ACTION TEST_CASE_3_EXEC:
                        IF vTestCases[2].state = utTestCaseStates.ut_RUNNING THEN
	(*Run the test case*)
	IF NOT assertGreaterEqual_DINT(vTestCase3_act, vTestCase3_xp) THEN
		vTestCases[2].state := utTestCaseStates.ut_PASSED;
		vTestCases[2].msg := 'Parameter act was less than xp and function returned FALSE -> PASS';
	ELSE
		vTestCases[2].state := utTestCaseStates.ut_FAILED;
		vTestCases[2].msg := 'Parameter act was less than xp and function returned TRUE -> FAIL';
	END_IF
END_IF
                      
END_ACTION
END_PROGRAM

PROGRAM test_assertGreaterEqual_LWORD
  VAR
    vTestCases : ARRAY[0..20] OF utTestCase;  (* Definition of all test cases for this POU *)
    testRunner : utTestSuite;  (* Test Suite fb instance to run the tests *)
    vRunAll : BOOL;  (* Manual command to run all tests for this POU *)
    vResetAll : BOOL;  (* Manual command to reset all tests for this POU *)
    vTestCase1_act : LWORD;  (* Test data 1 of test case 1 *)
    vTestCase1_xp : LWORD;  (* Test data 2 of test case 1 *)
    vTestCase2_act : LWORD;  (* Test data 1 of test case 2 *)
    vTestCase2_xp : LWORD;  (* Test data 2 of test case 2 *)
    vTestCase3_act : LWORD;  (* Test data 1 of test case 3 *)
    vTestCase3_xp : LWORD;  (* Test data 2 of test case 3 *)
  END_VAR

                    (*Run the test cases*)
TEST_CASE_1_SETUP();
TEST_CASE_1_EXEC();

TEST_CASE_2_SETUP();
TEST_CASE_2_EXEC();

TEST_CASE_3_SETUP();
TEST_CASE_3_EXEC();

(*Instantiate the test runner*)
testRunner(
	Id := 75,
	Name := 'assertGreaterEqual_LWORD',
    RunTests := GVL.RunAll OR vRunAll,
	ResetTests := GVL.ResetAll OR vResetAll,
	TestCases:=vTestCases);

(*Report the results to the collection global*)
GVL.Results[testRunner.Id] := testRunner.Summary;
                  

ACTION TEST_CASE_1_EXEC:
                        IF vTestCases[0].state = utTestCaseStates.ut_RUNNING THEN
	(*Run the test case*)
	IF assertGreaterEqual_LWORD(vTestCase1_act, vTestCase1_xp) THEN
		vTestCases[0].state := utTestCaseStates.ut_PASSED;
		vTestCases[0].msg := 'Parameter act was greater than xp and function returned TRUE -> PASS';
	ELSE
		vTestCases[0].state := utTestCaseStates.ut_FAILED;
		vTestCases[0].msg := 'Parameter act was greater than xp and function returned FALSE -> FAIL';
	END_IF
END_IF
                      
END_ACTION

ACTION TEST_CASE_3_EXEC:
                        IF vTestCases[2].state = utTestCaseStates.ut_RUNNING THEN
	(*Run the test case*)
	IF NOT assertGreaterEqual_LWORD(vTestCase3_act, vTestCase3_xp) THEN
		vTestCases[2].state := utTestCaseStates.ut_PASSED;
		vTestCases[2].msg := 'Parameter act was less than xp and function returned FALSE -> PASS';
	ELSE
		vTestCases[2].state := utTestCaseStates.ut_FAILED;
		vTestCases[2].msg := 'Parameter act was less than xp and function returned TRUE -> FAIL';
	END_IF
END_IF
                      
END_ACTION

ACTION TEST_CASE_1_SETUP:
                        IF vTestCases[0].state = utTestCaseStates.ut_SETUP THEN
	(*Setup the test case information*)
	vTestCases[0].id := 1;
	vTestCases[0].desc[0] := 'RETURNS TRUE WHEN PARAMETER ACT GREATER THAN XP';
    vTestCases[0].desc[1] := 'Tests if the function returns True if the parameter act is greater than parameter xp';
	vTestCases[0].desc[2] := 'PASS IF: Return value is TRUE';
	
	(*Setup needed variables*)
	vTestCase1_act := REAL_TO_LWORD(115.4);
	vTestCase1_xp := REAL_TO_LWORD(85.4);
END_IF
                      
END_ACTION

ACTION TEST_CASE_2_SETUP:
                        IF vTestCases[1].state = utTestCaseStates.ut_SETUP THEN
	(*Setup the test case information*)
	vTestCases[1].id := 2;
    vTestCases[1].desc[0] := 'RETURNS TRUE WHEN PARAMETER ACT EQUAL TO XP';
    vTestCases[1].desc[1] := 'Tests if the function returns True if the parameter act is equal to parameter xp';
	vTestCases[1].desc[2] := 'PASS IF: Return value is TRUE';
	
	(*Setup needed variables*)
	vTestCase2_act := REAL_TO_LWORD(115.4);
	vTestCase2_xp := REAL_TO_LWORD(115.4);
END_IF
                      
END_ACTION

ACTION TEST_CASE_2_EXEC:
                        IF vTestCases[1].state = utTestCaseStates.ut_RUNNING THEN
	(*Run the test case*)
	IF assertGreaterEqual_LWORD(vTestCase2_act, vTestCase2_xp) THEN
		vTestCases[1].state := utTestCaseStates.ut_PASSED;
		vTestCases[1].msg := 'Parameter act was equal to xp and function returned TRUE -> PASS';
	ELSE
		vTestCases[1].state := utTestCaseStates.ut_FAILED;
		vTestCases[1].msg := 'Parameter act was equal to xp and function returned FALSE -> FAIL';
	END_IF
END_IF
                      
END_ACTION

ACTION TEST_CASE_3_SETUP:
                        IF vTestCases[2].state = utTestCaseStates.ut_SETUP THEN
	(*Setup the test case information*)
	vTestCases[2].id := 3;
    vTestCases[2].desc[0] := 'RETURNS FALSE WHEN PARAMETER ACT LESS THAN XP';
    vTestCases[2].desc[1] := 'Tests if the function returns False if the parameter act is less than parameter xp';
	vTestCases[2].desc[2] := 'PASS IF: Return value is FALSE';
	
	(*Setup needed variables*)
	vTestCase3_act := REAL_TO_LWORD(85.4);
	vTestCase3_xp := REAL_TO_LWORD(115.4);
END_IF
                      
END_ACTION
END_PROGRAM

PROGRAM test_assertGreaterEqual_ULINT
  VAR
    vTestCases : ARRAY[0..20] OF utTestCase;  (* Definition of all test cases for this POU *)
    testRunner : utTestSuite;  (* Test Suite fb instance to run the tests *)
    vRunAll : BOOL;  (* Manual command to run all tests for this POU *)
    vResetAll : BOOL;  (* Manual command to reset all tests for this POU *)
    vTestCase1_act : ULINT;  (* Test data 1 of test case 1 *)
    vTestCase1_xp : ULINT;  (* Test data 2 of test case 1 *)
    vTestCase2_act : ULINT;  (* Test data 1 of test case 2 *)
    vTestCase2_xp : ULINT;  (* Test data 2 of test case 2 *)
    vTestCase3_act : ULINT;  (* Test data 1 of test case 3 *)
    vTestCase3_xp : ULINT;  (* Test data 2 of test case 3 *)
  END_VAR

                    (*Run the test cases*)
TEST_CASE_1_SETUP();
TEST_CASE_1_EXEC();

TEST_CASE_2_SETUP();
TEST_CASE_2_EXEC();

TEST_CASE_3_SETUP();
TEST_CASE_3_EXEC();

(*Instantiate the test runner*)
testRunner(
	Id := 83,
	Name := 'assertGreaterEqual_ULINT',
    RunTests := GVL.RunAll OR vRunAll,
	ResetTests := GVL.ResetAll OR vResetAll,
	TestCases:=vTestCases);

(*Report the results to the collection global*)
GVL.Results[testRunner.Id] := testRunner.Summary;
                  

ACTION TEST_CASE_2_EXEC:
                        IF vTestCases[1].state = utTestCaseStates.ut_RUNNING THEN
	(*Run the test case*)
	IF assertGreaterEqual_ULINT(vTestCase2_act, vTestCase2_xp) THEN
		vTestCases[1].state := utTestCaseStates.ut_PASSED;
		vTestCases[1].msg := 'Parameter act was equal to xp and function returned TRUE -> PASS';
	ELSE
		vTestCases[1].state := utTestCaseStates.ut_FAILED;
		vTestCases[1].msg := 'Parameter act was equal to xp and function returned FALSE -> FAIL';
	END_IF
END_IF
                      
END_ACTION

ACTION TEST_CASE_1_SETUP:
                        IF vTestCases[0].state = utTestCaseStates.ut_SETUP THEN
	(*Setup the test case information*)
	vTestCases[0].id := 1;
	vTestCases[0].desc[0] := 'RETURNS TRUE WHEN PARAMETER ACT GREATER THAN XP';
    vTestCases[0].desc[1] := 'Tests if the function returns True if the parameter act is greater than parameter xp';
	vTestCases[0].desc[2] := 'PASS IF: Return value is TRUE';
	
	(*Setup needed variables*)
	vTestCase1_act := REAL_TO_ULINT(115.4);
	vTestCase1_xp := REAL_TO_ULINT(85.4);
END_IF
                      
END_ACTION

ACTION TEST_CASE_1_EXEC:
                        IF vTestCases[0].state = utTestCaseStates.ut_RUNNING THEN
	(*Run the test case*)
	IF assertGreaterEqual_ULINT(vTestCase1_act, vTestCase1_xp) THEN
		vTestCases[0].state := utTestCaseStates.ut_PASSED;
		vTestCases[0].msg := 'Parameter act was greater than xp and function returned TRUE -> PASS';
	ELSE
		vTestCases[0].state := utTestCaseStates.ut_FAILED;
		vTestCases[0].msg := 'Parameter act was greater than xp and function returned FALSE -> FAIL';
	END_IF
END_IF
                      
END_ACTION

ACTION TEST_CASE_2_SETUP:
                        IF vTestCases[1].state = utTestCaseStates.ut_SETUP THEN
	(*Setup the test case information*)
	vTestCases[1].id := 2;
    vTestCases[1].desc[0] := 'RETURNS TRUE WHEN PARAMETER ACT EQUAL TO XP';
    vTestCases[1].desc[1] := 'Tests if the function returns True if the parameter act is equal to parameter xp';
	vTestCases[1].desc[2] := 'PASS IF: Return value is TRUE';
	
	(*Setup needed variables*)
	vTestCase2_act := REAL_TO_ULINT(115.4);
	vTestCase2_xp := REAL_TO_ULINT(115.4);
END_IF
                      
END_ACTION

ACTION TEST_CASE_3_SETUP:
                        IF vTestCases[2].state = utTestCaseStates.ut_SETUP THEN
	(*Setup the test case information*)
	vTestCases[2].id := 3;
    vTestCases[2].desc[0] := 'RETURNS FALSE WHEN PARAMETER ACT LESS THAN XP';
    vTestCases[2].desc[1] := 'Tests if the function returns False if the parameter act is less than parameter xp';
	vTestCases[2].desc[2] := 'PASS IF: Return value is FALSE';
	
	(*Setup needed variables*)
	vTestCase3_act := REAL_TO_ULINT(85.4);
	vTestCase3_xp := REAL_TO_ULINT(115.4);
END_IF
                      
END_ACTION

ACTION TEST_CASE_3_EXEC:
                        IF vTestCases[2].state = utTestCaseStates.ut_RUNNING THEN
	(*Run the test case*)
	IF NOT assertGreaterEqual_ULINT(vTestCase3_act, vTestCase3_xp) THEN
		vTestCases[2].state := utTestCaseStates.ut_PASSED;
		vTestCases[2].msg := 'Parameter act was less than xp and function returned FALSE -> PASS';
	ELSE
		vTestCases[2].state := utTestCaseStates.ut_FAILED;
		vTestCases[2].msg := 'Parameter act was less than xp and function returned TRUE -> FAIL';
	END_IF
END_IF
                      
END_ACTION
END_PROGRAM

PROGRAM test_assertGreaterEqual_SINT
  VAR
    vTestCases : ARRAY[0..20] OF utTestCase;  (* Definition of all test cases for this POU *)
    testRunner : utTestSuite;  (* Test Suite fb instance to run the tests *)
    vRunAll : BOOL;  (* Manual command to run all tests for this POU *)
    vResetAll : BOOL;  (* Manual command to reset all tests for this POU *)
    vTestCase1_act : SINT;  (* Test data 1 of test case 1 *)
    vTestCase1_xp : SINT;  (* Test data 2 of test case 1 *)
    vTestCase2_act : SINT;  (* Test data 1 of test case 2 *)
    vTestCase2_xp : SINT;  (* Test data 2 of test case 2 *)
    vTestCase3_act : SINT;  (* Test data 1 of test case 3 *)
    vTestCase3_xp : SINT;  (* Test data 2 of test case 3 *)
  END_VAR

                    (*Run the test cases*)
TEST_CASE_1_SETUP();
TEST_CASE_1_EXEC();

TEST_CASE_2_SETUP();
TEST_CASE_2_EXEC();

TEST_CASE_3_SETUP();
TEST_CASE_3_EXEC();

(*Instantiate the test runner*)
testRunner(
	Id := 76,
	Name := 'assertGreaterEqual_SINT',
    RunTests := GVL.RunAll OR vRunAll,
	ResetTests := GVL.ResetAll OR vResetAll,
	TestCases:=vTestCases);

(*Report the results to the collection global*)
GVL.Results[testRunner.Id] := testRunner.Summary;
                  

ACTION TEST_CASE_2_EXEC:
                        IF vTestCases[1].state = utTestCaseStates.ut_RUNNING THEN
	(*Run the test case*)
	IF assertGreaterEqual_SINT(vTestCase2_act, vTestCase2_xp) THEN
		vTestCases[1].state := utTestCaseStates.ut_PASSED;
		vTestCases[1].msg := 'Parameter act was equal to xp and function returned TRUE -> PASS';
	ELSE
		vTestCases[1].state := utTestCaseStates.ut_FAILED;
		vTestCases[1].msg := 'Parameter act was equal to xp and function returned FALSE -> FAIL';
	END_IF
END_IF
                      
END_ACTION

ACTION TEST_CASE_1_SETUP:
                        IF vTestCases[0].state = utTestCaseStates.ut_SETUP THEN
	(*Setup the test case information*)
	vTestCases[0].id := 1;
	vTestCases[0].desc[0] := 'RETURNS TRUE WHEN PARAMETER ACT GREATER THAN XP';
    vTestCases[0].desc[1] := 'Tests if the function returns True if the parameter act is greater than parameter xp';
	vTestCases[0].desc[2] := 'PASS IF: Return value is TRUE';
	
	(*Setup needed variables*)
	vTestCase1_act := REAL_TO_SINT(115.4);
	vTestCase1_xp := REAL_TO_SINT(85.4);
END_IF
                      
END_ACTION

ACTION TEST_CASE_1_EXEC:
                        IF vTestCases[0].state = utTestCaseStates.ut_RUNNING THEN
	(*Run the test case*)
	IF assertGreaterEqual_SINT(vTestCase1_act, vTestCase1_xp) THEN
		vTestCases[0].state := utTestCaseStates.ut_PASSED;
		vTestCases[0].msg := 'Parameter act was greater than xp and function returned TRUE -> PASS';
	ELSE
		vTestCases[0].state := utTestCaseStates.ut_FAILED;
		vTestCases[0].msg := 'Parameter act was greater than xp and function returned FALSE -> FAIL';
	END_IF
END_IF
                      
END_ACTION

ACTION TEST_CASE_2_SETUP:
                        IF vTestCases[1].state = utTestCaseStates.ut_SETUP THEN
	(*Setup the test case information*)
	vTestCases[1].id := 2;
    vTestCases[1].desc[0] := 'RETURNS TRUE WHEN PARAMETER ACT EQUAL TO XP';
    vTestCases[1].desc[1] := 'Tests if the function returns True if the parameter act is equal to parameter xp';
	vTestCases[1].desc[2] := 'PASS IF: Return value is TRUE';
	
	(*Setup needed variables*)
	vTestCase2_act := REAL_TO_SINT(115.4);
	vTestCase2_xp := REAL_TO_SINT(115.4);
END_IF
                      
END_ACTION

ACTION TEST_CASE_3_SETUP:
                        IF vTestCases[2].state = utTestCaseStates.ut_SETUP THEN
	(*Setup the test case information*)
	vTestCases[2].id := 3;
    vTestCases[2].desc[0] := 'RETURNS FALSE WHEN PARAMETER ACT LESS THAN XP';
    vTestCases[2].desc[1] := 'Tests if the function returns False if the parameter act is less than parameter xp';
	vTestCases[2].desc[2] := 'PASS IF: Return value is FALSE';
	
	(*Setup needed variables*)
	vTestCase3_act := REAL_TO_SINT(85.4);
	vTestCase3_xp := REAL_TO_SINT(115.4);
END_IF
                      
END_ACTION

ACTION TEST_CASE_3_EXEC:
                        IF vTestCases[2].state = utTestCaseStates.ut_RUNNING THEN
	(*Run the test case*)
	IF NOT assertGreaterEqual_SINT(vTestCase3_act, vTestCase3_xp) THEN
		vTestCases[2].state := utTestCaseStates.ut_PASSED;
		vTestCases[2].msg := 'Parameter act was less than xp and function returned FALSE -> PASS';
	ELSE
		vTestCases[2].state := utTestCaseStates.ut_FAILED;
		vTestCases[2].msg := 'Parameter act was less than xp and function returned TRUE -> FAIL';
	END_IF
END_IF
                      
END_ACTION
END_PROGRAM

PROGRAM test_assertGreater_LREAL
  VAR
    vTestCases : ARRAY[0..20] OF utTestCase;  (* Definition of all test cases for this POU *)
    testRunner : utTestSuite;  (* Test Suite fb instance to run the tests *)
    vRunAll : BOOL;  (* Manual command to run all tests for this POU *)
    vResetAll : BOOL;  (* Manual command to reset all tests for this POU *)
    vTestCase1_act : LREAL;  (* Test data 1 of test case 1 *)
    vTestCase1_xp : LREAL;  (* Test data 2 of test case 1 *)
    vTestCase2_act : LREAL;  (* Test data 1 of test case 2 *)
    vTestCase2_xp : LREAL;  (* Test data 2 of test case 2 *)
  END_VAR

                    (*Run the test cases*)
TEST_CASE_1_SETUP();
TEST_CASE_1_EXEC();

TEST_CASE_2_SETUP();
TEST_CASE_2_EXEC();

(*Instantiate the test runner*)
testRunner(
	Id := 63,
	Name := 'assertGreater_LREAL',
    RunTests := GVL.RunAll OR vRunAll,
	ResetTests := GVL.ResetAll OR vResetAll,
	TestCases:=vTestCases);

(*Report the results to the collection global*)
GVL.Results[testRunner.Id] := testRunner.Summary;
                  

ACTION TEST_CASE_1_SETUP:
                        IF vTestCases[0].state = utTestCaseStates.ut_SETUP THEN
	(*Setup the test case information*)
	vTestCases[0].id := 1;
	vTestCases[0].desc[0] := 'RETURNS TRUE WHEN PARAMETER ACT GREATER THAN XP';
    vTestCases[0].desc[1] := 'Tests if the function returns True if the parameter act is greater than parameter xp';
	vTestCases[0].desc[2] := 'PASS IF: Return value is TRUE';
	
	(*Setup needed variables*)
	vTestCase1_act := REAL_TO_LREAL(115.4);
	vTestCase1_xp := REAL_TO_LREAL(85.4);
END_IF
                      
END_ACTION

ACTION TEST_CASE_1_EXEC:
                        IF vTestCases[0].state = utTestCaseStates.ut_RUNNING THEN
	(*Run the test case*)
	IF assertGreater_LREAL(vTestCase1_act, vTestCase1_xp) THEN
		vTestCases[0].state := utTestCaseStates.ut_PASSED;
		vTestCases[0].msg := 'Parameter act was greater than xp and function returned TRUE -> PASS';
	ELSE
		vTestCases[0].state := utTestCaseStates.ut_FAILED;
		vTestCases[0].msg := 'Parameter act was greater than xp and function returned FALSE -> FAIL';
	END_IF
END_IF
                      
END_ACTION

ACTION TEST_CASE_2_SETUP:
                        IF vTestCases[1].state = utTestCaseStates.ut_SETUP THEN
	(*Setup the test case information*)
	vTestCases[1].id := 2;
    vTestCases[1].desc[0] := 'RETURNS FALSE WHEN PARAMETER ACT LESS THAN XP';
    vTestCases[1].desc[1] := 'Tests if the function returns False if the parameter act is less than parameter xp';
	vTestCases[1].desc[2] := 'PASS IF: Return value is FALSE';
	
	(*Setup needed variables*)
	vTestCase2_act := REAL_TO_LREAL(8.4);
	vTestCase2_xp := REAL_TO_LREAL(85.4);
END_IF
                      
END_ACTION

ACTION TEST_CASE_2_EXEC:
                        IF vTestCases[1].state = utTestCaseStates.ut_RUNNING THEN
	(*Run the test case*)
	IF NOT assertGreater_LREAL(vTestCase2_act, vTestCase2_xp) THEN
		vTestCases[1].state := utTestCaseStates.ut_PASSED;
		vTestCases[1].msg := 'Parameter act was less than xp and function returned FALSE -> PASS';
	ELSE
		vTestCases[1].state := utTestCaseStates.ut_FAILED;
		vTestCases[1].msg := 'Parameter act was less than xp and function returned TRUE -> FAIL';
	END_IF
END_IF
                      
END_ACTION
END_PROGRAM

PROGRAM test_assertGreater_TIME
  VAR
    vTestCases : ARRAY[0..20] OF utTestCase;  (* Definition of all test cases for this POU *)
    testRunner : utTestSuite;  (* Test Suite fb instance to run the tests *)
    vRunAll : BOOL;  (* Manual command to run all tests for this POU *)
    vResetAll : BOOL;  (* Manual command to reset all tests for this POU *)
    vTestCase1_act : TIME;  (* Test data 1 of test case 1 *)
    vTestCase1_xp : TIME;  (* Test data 2 of test case 1 *)
    vTestCase2_act : TIME;  (* Test data 1 of test case 2 *)
    vTestCase2_xp : TIME;  (* Test data 2 of test case 2 *)
  END_VAR

                    (*Run the test cases*)
TEST_CASE_1_SETUP();
TEST_CASE_1_EXEC();

TEST_CASE_2_SETUP();
TEST_CASE_2_EXEC();

(*Instantiate the test runner*)
testRunner(
	Id := 64,
	Name := 'assertGreater_TIME',
    RunTests := GVL.RunAll OR vRunAll,
	ResetTests := GVL.ResetAll OR vResetAll,
	TestCases:=vTestCases);

(*Report the results to the collection global*)
GVL.Results[testRunner.Id] := testRunner.Summary;
                  

ACTION TEST_CASE_1_SETUP:
                        IF vTestCases[0].state = utTestCaseStates.ut_SETUP THEN
	(*Setup the test case information*)
	vTestCases[0].id := 1;
	vTestCases[0].desc[0] := 'RETURNS TRUE WHEN PARAMETER ACT GREATER THAN XP';
    vTestCases[0].desc[1] := 'Tests if the function returns True if the parameter act is greater than parameter xp';
	vTestCases[0].desc[2] := 'PASS IF: Return value is TRUE';
	
	(*Setup needed variables*)
	vTestCase1_act := REAL_TO_TIME(115.4);
	vTestCase1_xp := REAL_TO_TIME(85.4);
END_IF
                      
END_ACTION

ACTION TEST_CASE_1_EXEC:
                        IF vTestCases[0].state = utTestCaseStates.ut_RUNNING THEN
	(*Run the test case*)
	IF assertGreater_TIME(vTestCase1_act, vTestCase1_xp) THEN
		vTestCases[0].state := utTestCaseStates.ut_PASSED;
		vTestCases[0].msg := 'Parameter act was greater than xp and function returned TRUE -> PASS';
	ELSE
		vTestCases[0].state := utTestCaseStates.ut_FAILED;
		vTestCases[0].msg := 'Parameter act was greater than xp and function returned FALSE -> FAIL';
	END_IF
END_IF
                      
END_ACTION

ACTION TEST_CASE_2_SETUP:
                        IF vTestCases[1].state = utTestCaseStates.ut_SETUP THEN
	(*Setup the test case information*)
	vTestCases[1].id := 2;
    vTestCases[1].desc[0] := 'RETURNS FALSE WHEN PARAMETER ACT LESS THAN XP';
    vTestCases[1].desc[1] := 'Tests if the function returns False if the parameter act is less than parameter xp';
	vTestCases[1].desc[2] := 'PASS IF: Return value is FALSE';
	
	(*Setup needed variables*)
	vTestCase2_act := REAL_TO_TIME(8.4);
	vTestCase2_xp := REAL_TO_TIME(85.4);
END_IF
                      
END_ACTION

ACTION TEST_CASE_2_EXEC:
                        IF vTestCases[1].state = utTestCaseStates.ut_RUNNING THEN
	(*Run the test case*)
	IF NOT assertGreater_TIME(vTestCase2_act, vTestCase2_xp) THEN
		vTestCases[1].state := utTestCaseStates.ut_PASSED;
		vTestCases[1].msg := 'Parameter act was less than xp and function returned FALSE -> PASS';
	ELSE
		vTestCases[1].state := utTestCaseStates.ut_FAILED;
		vTestCases[1].msg := 'Parameter act was less than xp and function returned TRUE -> FAIL';
	END_IF
END_IF
                      
END_ACTION
END_PROGRAM

PROGRAM test_assertGreater_TIME_OF_DAY
  VAR
    vTestCases : ARRAY[0..20] OF utTestCase;  (* Definition of all test cases for this POU *)
    testRunner : utTestSuite;  (* Test Suite fb instance to run the tests *)
    vRunAll : BOOL;  (* Manual command to run all tests for this POU *)
    vResetAll : BOOL;  (* Manual command to reset all tests for this POU *)
    vTestCase1_act : TOD;  (* Test data 1 of test case 1 *)
    vTestCase1_xp : TOD;  (* Test data 2 of test case 1 *)
    vTestCase2_act : TOD;  (* Test data 1 of test case 2 *)
    vTestCase2_xp : TOD;  (* Test data 2 of test case 2 *)
  END_VAR

                    (*Run the test cases*)
TEST_CASE_1_SETUP();
TEST_CASE_1_EXEC();

TEST_CASE_2_SETUP();
TEST_CASE_2_EXEC();

(*Instantiate the test runner*)
testRunner(
	Id := 70,
	Name := 'assertGreater_TIME_OF_DAY',
    RunTests := GVL.RunAll OR vRunAll,
	ResetTests := GVL.ResetAll OR vResetAll,
	TestCases:=vTestCases);

(*Report the results to the collection global*)
GVL.Results[testRunner.Id] := testRunner.Summary;
                  

ACTION TEST_CASE_1_SETUP:
                        IF vTestCases[0].state = utTestCaseStates.ut_SETUP THEN
	(*Setup the test case information*)
	vTestCases[0].id := 1;
	vTestCases[0].desc[0] := 'RETURNS TRUE WHEN PARAMETER ACT GREATER THAN XP';
    vTestCases[0].desc[1] := 'Tests if the function returns True if the parameter act is greater than parameter xp';
	vTestCases[0].desc[2] := 'PASS IF: Return value is TRUE';
	
	(*Setup needed variables*)
	vTestCase1_act := REAL_TO_TOD(115.4);
	vTestCase1_xp := REAL_TO_TOD(85.4);
END_IF
                      
END_ACTION

ACTION TEST_CASE_1_EXEC:
                        IF vTestCases[0].state = utTestCaseStates.ut_RUNNING THEN
	(*Run the test case*)
	IF assertGreater_TIME_OF_DAY(vTestCase1_act, vTestCase1_xp) THEN
		vTestCases[0].state := utTestCaseStates.ut_PASSED;
		vTestCases[0].msg := 'Parameter act was greater than xp and function returned TRUE -> PASS';
	ELSE
		vTestCases[0].state := utTestCaseStates.ut_FAILED;
		vTestCases[0].msg := 'Parameter act was greater than xp and function returned FALSE -> FAIL';
	END_IF
END_IF
                      
END_ACTION

ACTION TEST_CASE_2_SETUP:
                        IF vTestCases[1].state = utTestCaseStates.ut_SETUP THEN
	(*Setup the test case information*)
	vTestCases[1].id := 2;
    vTestCases[1].desc[0] := 'RETURNS FALSE WHEN PARAMETER ACT LESS THAN XP';
    vTestCases[1].desc[1] := 'Tests if the function returns False if the parameter act is less than parameter xp';
	vTestCases[1].desc[2] := 'PASS IF: Return value is FALSE';
	
	(*Setup needed variables*)
	vTestCase2_act := REAL_TO_TOD(8.4);
	vTestCase2_xp := REAL_TO_TOD(85.4);
END_IF
                      
END_ACTION

ACTION TEST_CASE_2_EXEC:
                        IF vTestCases[1].state = utTestCaseStates.ut_RUNNING THEN
	(*Run the test case*)
	IF NOT assertGreater_TIME_OF_DAY(vTestCase2_act, vTestCase2_xp) THEN
		vTestCases[1].state := utTestCaseStates.ut_PASSED;
		vTestCases[1].msg := 'Parameter act was less than xp and function returned FALSE -> PASS';
	ELSE
		vTestCases[1].state := utTestCaseStates.ut_FAILED;
		vTestCases[1].msg := 'Parameter act was less than xp and function returned TRUE -> FAIL';
	END_IF
END_IF
                      
END_ACTION
END_PROGRAM

PROGRAM test_assertGreater_LTIME_OF_DAY
  VAR
    vTestCases : ARRAY[0..20] OF utTestCase;  (* Definition of all test cases for this POU *)
    testRunner : utTestSuite;  (* Test Suite fb instance to run the tests *)
    vRunAll : BOOL;  (* Manual command to run all tests for this POU *)
    vResetAll : BOOL;  (* Manual command to reset all tests for this POU *)
    vTestCase1_act : LTIME_OF_DAY;  (* Test data 1 of test case 1 *)
    vTestCase1_xp : LTIME_OF_DAY;  (* Test data 2 of test case 1 *)
    vTestCase2_act : LTIME_OF_DAY;  (* Test data 1 of test case 2 *)
    vTestCase2_xp : LTIME_OF_DAY;  (* Test data 2 of test case 2 *)
  END_VAR

                    (*Run the test cases*)
TEST_CASE_1_SETUP();
TEST_CASE_1_EXEC();

TEST_CASE_2_SETUP();
TEST_CASE_2_EXEC();

(*Instantiate the test runner*)
testRunner(
	Id := 71,
	Name := 'assertGreater_LTIME_OF_DAY',
    RunTests := GVL.RunAll OR vRunAll,
	ResetTests := GVL.ResetAll OR vResetAll,
	TestCases:=vTestCases);

(*Report the results to the collection global*)
GVL.Results[testRunner.Id] := testRunner.Summary;
                  

ACTION TEST_CASE_1_SETUP:
                        IF vTestCases[0].state = utTestCaseStates.ut_SETUP THEN
	(*Setup the test case information*)
	vTestCases[0].id := 1;
	vTestCases[0].desc[0] := 'RETURNS TRUE WHEN PARAMETER ACT GREATER THAN XP';
    vTestCases[0].desc[1] := 'Tests if the function returns True if the parameter act is greater than parameter xp';
	vTestCases[0].desc[2] := 'PASS IF: Return value is TRUE';
	
	(*Setup needed variables*)
	vTestCase1_act := REAL_TO_LTOD(115.4);
	vTestCase1_xp := REAL_TO_LTOD(85.4);
END_IF
                      
END_ACTION

ACTION TEST_CASE_1_EXEC:
                        IF vTestCases[0].state = utTestCaseStates.ut_RUNNING THEN
	(*Run the test case*)
	IF assertGreater_LTIME_OF_DAY(vTestCase1_act, vTestCase1_xp) THEN
		vTestCases[0].state := utTestCaseStates.ut_PASSED;
		vTestCases[0].msg := 'Parameter act was greater than xp and function returned TRUE -> PASS';
	ELSE
		vTestCases[0].state := utTestCaseStates.ut_FAILED;
		vTestCases[0].msg := 'Parameter act was greater than xp and function returned FALSE -> FAIL';
	END_IF
END_IF
                      
END_ACTION

ACTION TEST_CASE_2_SETUP:
                        IF vTestCases[1].state = utTestCaseStates.ut_SETUP THEN
	(*Setup the test case information*)
	vTestCases[1].id := 2;
    vTestCases[1].desc[0] := 'RETURNS FALSE WHEN PARAMETER ACT LESS THAN XP';
    vTestCases[1].desc[1] := 'Tests if the function returns False if the parameter act is less than parameter xp';
	vTestCases[1].desc[2] := 'PASS IF: Return value is FALSE';
	
	(*Setup needed variables*)
	vTestCase2_act := REAL_TO_LTOD(8.4);
	vTestCase2_xp := REAL_TO_LTOD(85.4);
END_IF
                      
END_ACTION

ACTION TEST_CASE_2_EXEC:
                        IF vTestCases[1].state = utTestCaseStates.ut_RUNNING THEN
	(*Run the test case*)
	IF NOT assertGreater_LTIME_OF_DAY(vTestCase2_act, vTestCase2_xp) THEN
		vTestCases[1].state := utTestCaseStates.ut_PASSED;
		vTestCases[1].msg := 'Parameter act was less than xp and function returned FALSE -> PASS';
	ELSE
		vTestCases[1].state := utTestCaseStates.ut_FAILED;
		vTestCases[1].msg := 'Parameter act was less than xp and function returned TRUE -> FAIL';
	END_IF
END_IF
                      
END_ACTION
END_PROGRAM

PROGRAM test_assertGreater_LTIME
  VAR
    vTestCases : ARRAY[0..20] OF utTestCase;  (* Definition of all test cases for this POU *)
    testRunner : utTestSuite;  (* Test Suite fb instance to run the tests *)
    vRunAll : BOOL;  (* Manual command to run all tests for this POU *)
    vResetAll : BOOL;  (* Manual command to reset all tests for this POU *)
    vTestCase1_act : LTIME;  (* Test data 1 of test case 1 *)
    vTestCase1_xp : LTIME;  (* Test data 2 of test case 1 *)
    vTestCase2_act : LTIME;  (* Test data 1 of test case 2 *)
    vTestCase2_xp : LTIME;  (* Test data 2 of test case 2 *)
  END_VAR

                    (*Run the test cases*)
TEST_CASE_1_SETUP();
TEST_CASE_1_EXEC();

TEST_CASE_2_SETUP();
TEST_CASE_2_EXEC();

(*Instantiate the test runner*)
testRunner(
	Id := 65,
	Name := 'assertGreater_LTIME',
    RunTests := GVL.RunAll OR vRunAll,
	ResetTests := GVL.ResetAll OR vResetAll,
	TestCases:=vTestCases);

(*Report the results to the collection global*)
GVL.Results[testRunner.Id] := testRunner.Summary;
                  

ACTION TEST_CASE_2_SETUP:
                        IF vTestCases[1].state = utTestCaseStates.ut_SETUP THEN
	(*Setup the test case information*)
	vTestCases[1].id := 2;
    vTestCases[1].desc[0] := 'RETURNS FALSE WHEN PARAMETER ACT LESS THAN XP';
    vTestCases[1].desc[1] := 'Tests if the function returns False if the parameter act is less than parameter xp';
	vTestCases[1].desc[2] := 'PASS IF: Return value is FALSE';
	
	(*Setup needed variables*)
	vTestCase2_act := REAL_TO_LTIME(8.4);
	vTestCase2_xp := REAL_TO_LTIME(85.4);
END_IF
                      
END_ACTION

ACTION TEST_CASE_2_EXEC:
                        IF vTestCases[1].state = utTestCaseStates.ut_RUNNING THEN
	(*Run the test case*)
	IF NOT assertGreater_LTIME(vTestCase2_act, vTestCase2_xp) THEN
		vTestCases[1].state := utTestCaseStates.ut_PASSED;
		vTestCases[1].msg := 'Parameter act was less than xp and function returned FALSE -> PASS';
	ELSE
		vTestCases[1].state := utTestCaseStates.ut_FAILED;
		vTestCases[1].msg := 'Parameter act was less than xp and function returned TRUE -> FAIL';
	END_IF
END_IF
                      
END_ACTION

ACTION TEST_CASE_1_SETUP:
                        IF vTestCases[0].state = utTestCaseStates.ut_SETUP THEN
	(*Setup the test case information*)
	vTestCases[0].id := 1;
	vTestCases[0].desc[0] := 'RETURNS TRUE WHEN PARAMETER ACT GREATER THAN XP';
    vTestCases[0].desc[1] := 'Tests if the function returns True if the parameter act is greater than parameter xp';
	vTestCases[0].desc[2] := 'PASS IF: Return value is TRUE';
	
	(*Setup needed variables*)
	vTestCase1_act := REAL_TO_LTIME(115.4);
	vTestCase1_xp := REAL_TO_LTIME(85.4);
END_IF
                      
END_ACTION

ACTION TEST_CASE_1_EXEC:
                        IF vTestCases[0].state = utTestCaseStates.ut_RUNNING THEN
	(*Run the test case*)
	IF assertGreater_LTIME(vTestCase1_act, vTestCase1_xp) THEN
		vTestCases[0].state := utTestCaseStates.ut_PASSED;
		vTestCases[0].msg := 'Parameter act was greater than xp and function returned TRUE -> PASS';
	ELSE
		vTestCases[0].state := utTestCaseStates.ut_FAILED;
		vTestCases[0].msg := 'Parameter act was greater than xp and function returned FALSE -> FAIL';
	END_IF
END_IF
                      
END_ACTION
END_PROGRAM

PROGRAM test_assertGreaterEqual_BYTE
  VAR
    vTestCases : ARRAY[0..20] OF utTestCase;  (* Definition of all test cases for this POU *)
    testRunner : utTestSuite;  (* Test Suite fb instance to run the tests *)
    vRunAll : BOOL;  (* Manual command to run all tests for this POU *)
    vResetAll : BOOL;  (* Manual command to reset all tests for this POU *)
    vTestCase1_act : BYTE;  (* Test data 1 of test case 1 *)
    vTestCase1_xp : BYTE;  (* Test data 2 of test case 1 *)
    vTestCase2_act : BYTE;  (* Test data 1 of test case 2 *)
    vTestCase2_xp : BYTE;  (* Test data 2 of test case 2 *)
    vTestCase3_act : BYTE;  (* Test data 1 of test case 3 *)
    vTestCase3_xp : BYTE;  (* Test data 2 of test case 3 *)
  END_VAR

                    (*Run the test cases*)
TEST_CASE_1_SETUP();
TEST_CASE_1_EXEC();

TEST_CASE_2_SETUP();
TEST_CASE_2_EXEC();

TEST_CASE_3_SETUP();
TEST_CASE_3_EXEC();

(*Instantiate the test runner*)
testRunner(
	Id := 72,
	Name := 'assertGreaterEqual_BYTE',
    RunTests := GVL.RunAll OR vRunAll,
	ResetTests := GVL.ResetAll OR vResetAll,
	TestCases:=vTestCases);

(*Report the results to the collection global*)
GVL.Results[testRunner.Id] := testRunner.Summary;
                  

ACTION TEST_CASE_2_SETUP:
                        IF vTestCases[1].state = utTestCaseStates.ut_SETUP THEN
	(*Setup the test case information*)
	vTestCases[1].id := 2;
    vTestCases[1].desc[0] := 'RETURNS TRUE WHEN PARAMETER ACT EQUAL TO XP';
    vTestCases[1].desc[1] := 'Tests if the function returns True if the parameter act is equal to parameter xp';
	vTestCases[1].desc[2] := 'PASS IF: Return value is TRUE';
	
	(*Setup needed variables*)
	vTestCase2_act := REAL_TO_BYTE(115.4);
	vTestCase2_xp := REAL_TO_BYTE(115.4);
END_IF
                      
END_ACTION

ACTION TEST_CASE_3_SETUP:
                        IF vTestCases[2].state = utTestCaseStates.ut_SETUP THEN
	(*Setup the test case information*)
	vTestCases[2].id := 3;
    vTestCases[2].desc[0] := 'RETURNS FALSE WHEN PARAMETER ACT LESS THAN XP';
    vTestCases[2].desc[1] := 'Tests if the function returns False if the parameter act is less than parameter xp';
	vTestCases[2].desc[2] := 'PASS IF: Return value is FALSE';
	
	(*Setup needed variables*)
	vTestCase3_act := REAL_TO_BYTE(85.4);
	vTestCase3_xp := REAL_TO_BYTE(115.4);
END_IF
                      
END_ACTION

ACTION TEST_CASE_2_EXEC:
                        IF vTestCases[1].state = utTestCaseStates.ut_RUNNING THEN
	(*Run the test case*)
	IF assertGreaterEqual_BYTE(vTestCase2_act, vTestCase2_xp) THEN
		vTestCases[1].state := utTestCaseStates.ut_PASSED;
		vTestCases[1].msg := 'Parameter act was equal to xp and function returned TRUE -> PASS';
	ELSE
		vTestCases[1].state := utTestCaseStates.ut_FAILED;
		vTestCases[1].msg := 'Parameter act was equal to xp and function returned FALSE -> FAIL';
	END_IF
END_IF
                      
END_ACTION

ACTION TEST_CASE_1_SETUP:
                        IF vTestCases[0].state = utTestCaseStates.ut_SETUP THEN
	(*Setup the test case information*)
	vTestCases[0].id := 1;
	vTestCases[0].desc[0] := 'RETURNS TRUE WHEN PARAMETER ACT GREATER THAN XP';
    vTestCases[0].desc[1] := 'Tests if the function returns True if the parameter act is greater than parameter xp';
	vTestCases[0].desc[2] := 'PASS IF: Return value is TRUE';
	
	(*Setup needed variables*)
	vTestCase1_act := REAL_TO_BYTE(115.4);
	vTestCase1_xp := REAL_TO_BYTE(85.4);
END_IF
                      
END_ACTION

ACTION TEST_CASE_1_EXEC:
                        IF vTestCases[0].state = utTestCaseStates.ut_RUNNING THEN
	(*Run the test case*)
	IF assertGreaterEqual_BYTE(vTestCase1_act, vTestCase1_xp) THEN
		vTestCases[0].state := utTestCaseStates.ut_PASSED;
		vTestCases[0].msg := 'Parameter act was greater than xp and function returned TRUE -> PASS';
	ELSE
		vTestCases[0].state := utTestCaseStates.ut_FAILED;
		vTestCases[0].msg := 'Parameter act was greater than xp and function returned FALSE -> FAIL';
	END_IF
END_IF
                      
END_ACTION

ACTION TEST_CASE_3_EXEC:
                        IF vTestCases[2].state = utTestCaseStates.ut_RUNNING THEN
	(*Run the test case*)
	IF NOT assertGreaterEqual_BYTE(vTestCase3_act, vTestCase3_xp) THEN
		vTestCases[2].state := utTestCaseStates.ut_PASSED;
		vTestCases[2].msg := 'Parameter act was less than xp and function returned FALSE -> PASS';
	ELSE
		vTestCases[2].state := utTestCaseStates.ut_FAILED;
		vTestCases[2].msg := 'Parameter act was less than xp and function returned TRUE -> FAIL';
	END_IF
END_IF
                      
END_ACTION
END_PROGRAM

PROGRAM test_assertGreaterEqual_REAL
  VAR
    vTestCases : ARRAY[0..20] OF utTestCase;  (* Definition of all test cases for this POU *)
    testRunner : utTestSuite;  (* Test Suite fb instance to run the tests *)
    vRunAll : BOOL;  (* Manual command to run all tests for this POU *)
    vResetAll : BOOL;  (* Manual command to reset all tests for this POU *)
    vTestCase1_act : REAL;  (* Test data 1 of test case 1 *)
    vTestCase1_xp : REAL;  (* Test data 2 of test case 1 *)
    vTestCase2_act : REAL;  (* Test data 1 of test case 2 *)
    vTestCase2_xp : REAL;  (* Test data 2 of test case 2 *)
    vTestCase3_act : REAL;  (* Test data 1 of test case 3 *)
    vTestCase3_xp : REAL;  (* Test data 2 of test case 3 *)
  END_VAR

                    (*Run the test cases*)
TEST_CASE_1_SETUP();
TEST_CASE_1_EXEC();

TEST_CASE_2_SETUP();
TEST_CASE_2_EXEC();

TEST_CASE_3_SETUP();
TEST_CASE_3_EXEC();

(*Instantiate the test runner*)
testRunner(
	Id := 84,
	Name := 'assertGreaterEqual_REAL',
    RunTests := GVL.RunAll OR vRunAll,
	ResetTests := GVL.ResetAll OR vResetAll,
	TestCases:=vTestCases);

(*Report the results to the collection global*)
GVL.Results[testRunner.Id] := testRunner.Summary;
                  

ACTION TEST_CASE_1_SETUP:
                        IF vTestCases[0].state = utTestCaseStates.ut_SETUP THEN
	(*Setup the test case information*)
	vTestCases[0].id := 1;
	vTestCases[0].desc[0] := 'RETURNS TRUE WHEN PARAMETER ACT GREATER THAN XP';
    vTestCases[0].desc[1] := 'Tests if the function returns True if the parameter act is greater than parameter xp';
	vTestCases[0].desc[2] := 'PASS IF: Return value is TRUE';
	
	(*Setup needed variables*)
	vTestCase1_act := 115.4;
	vTestCase1_xp := 85.4;
END_IF
                      
END_ACTION

ACTION TEST_CASE_1_EXEC:
                        IF vTestCases[0].state = utTestCaseStates.ut_RUNNING THEN
	(*Run the test case*)
	IF assertGreaterEqual_REAL(vTestCase1_act, vTestCase1_xp) THEN
		vTestCases[0].state := utTestCaseStates.ut_PASSED;
		vTestCases[0].msg := 'Parameter act was greater than xp and function returned TRUE -> PASS';
	ELSE
		vTestCases[0].state := utTestCaseStates.ut_FAILED;
		vTestCases[0].msg := 'Parameter act was greater than xp and function returned FALSE -> FAIL';
	END_IF
END_IF
                      
END_ACTION

ACTION TEST_CASE_2_SETUP:
                        IF vTestCases[1].state = utTestCaseStates.ut_SETUP THEN
	(*Setup the test case information*)
	vTestCases[1].id := 2;
    vTestCases[1].desc[0] := 'RETURNS TRUE WHEN PARAMETER ACT EQUAL TO XP';
    vTestCases[1].desc[1] := 'Tests if the function returns True if the parameter act is equal to parameter xp';
	vTestCases[1].desc[2] := 'PASS IF: Return value is TRUE';
	
	(*Setup needed variables*)
	vTestCase2_act := 115.4;
	vTestCase2_xp := 115.4;
END_IF
                      
END_ACTION

ACTION TEST_CASE_2_EXEC:
                        IF vTestCases[1].state = utTestCaseStates.ut_RUNNING THEN
	(*Run the test case*)
	IF assertGreaterEqual_REAL(vTestCase2_act, vTestCase2_xp) THEN
		vTestCases[1].state := utTestCaseStates.ut_PASSED;
		vTestCases[1].msg := 'Parameter act was equal to xp and function returned TRUE -> PASS';
	ELSE
		vTestCases[1].state := utTestCaseStates.ut_FAILED;
		vTestCases[1].msg := 'Parameter act was equal to xp and function returned FALSE -> FAIL';
	END_IF
END_IF
                      
END_ACTION

ACTION TEST_CASE_3_SETUP:
                        IF vTestCases[2].state = utTestCaseStates.ut_SETUP THEN
	(*Setup the test case information*)
	vTestCases[2].id := 3;
    vTestCases[2].desc[0] := 'RETURNS FALSE WHEN PARAMETER ACT LESS THAN XP';
    vTestCases[2].desc[1] := 'Tests if the function returns False if the parameter act is less than parameter xp';
	vTestCases[2].desc[2] := 'PASS IF: Return value is FALSE';
	
	(*Setup needed variables*)
	vTestCase3_act := 85.4;
	vTestCase3_xp := 115.4;
END_IF
                      
END_ACTION

ACTION TEST_CASE_3_EXEC:
                        IF vTestCases[2].state = utTestCaseStates.ut_RUNNING THEN
	(*Run the test case*)
	IF NOT assertGreaterEqual_REAL(vTestCase3_act, vTestCase3_xp) THEN
		vTestCases[2].state := utTestCaseStates.ut_PASSED;
		vTestCases[2].msg := 'Parameter act was less than xp and function returned FALSE -> PASS';
	ELSE
		vTestCases[2].state := utTestCaseStates.ut_FAILED;
		vTestCases[2].msg := 'Parameter act was less than xp and function returned TRUE -> FAIL';
	END_IF
END_IF
                      
END_ACTION
END_PROGRAM

PROGRAM test_assertGreaterEqual_LREAL
  VAR
    vTestCases : ARRAY[0..20] OF utTestCase;  (* Definition of all test cases for this POU *)
    testRunner : utTestSuite;  (* Test Suite fb instance to run the tests *)
    vRunAll : BOOL;  (* Manual command to run all tests for this POU *)
    vResetAll : BOOL;  (* Manual command to reset all tests for this POU *)
    vTestCase1_act : LREAL;  (* Test data 1 of test case 1 *)
    vTestCase1_xp : LREAL;  (* Test data 2 of test case 1 *)
    vTestCase2_act : LREAL;  (* Test data 1 of test case 2 *)
    vTestCase2_xp : LREAL;  (* Test data 2 of test case 2 *)
    vTestCase3_act : LREAL;  (* Test data 1 of test case 3 *)
    vTestCase3_xp : LREAL;  (* Test data 2 of test case 3 *)
  END_VAR

                    (*Run the test cases*)
TEST_CASE_1_SETUP();
TEST_CASE_1_EXEC();

TEST_CASE_2_SETUP();
TEST_CASE_2_EXEC();

TEST_CASE_3_SETUP();
TEST_CASE_3_EXEC();

(*Instantiate the test runner*)
testRunner(
	Id := 85,
	Name := 'assertGreaterEqual_LREAL',
    RunTests := GVL.RunAll OR vRunAll,
	ResetTests := GVL.ResetAll OR vResetAll,
	TestCases:=vTestCases);

(*Report the results to the collection global*)
GVL.Results[testRunner.Id] := testRunner.Summary;
                  

ACTION TEST_CASE_1_SETUP:
                        IF vTestCases[0].state = utTestCaseStates.ut_SETUP THEN
	(*Setup the test case information*)
	vTestCases[0].id := 1;
	vTestCases[0].desc[0] := 'RETURNS TRUE WHEN PARAMETER ACT GREATER THAN XP';
    vTestCases[0].desc[1] := 'Tests if the function returns True if the parameter act is greater than parameter xp';
	vTestCases[0].desc[2] := 'PASS IF: Return value is TRUE';
	
	(*Setup needed variables*)
	vTestCase1_act := REAL_TO_LREAL(115.4);
	vTestCase1_xp := REAL_TO_LREAL(85.4);
END_IF
                      
END_ACTION

ACTION TEST_CASE_1_EXEC:
                        IF vTestCases[0].state = utTestCaseStates.ut_RUNNING THEN
	(*Run the test case*)
	IF assertGreaterEqual_LREAL(vTestCase1_act, vTestCase1_xp) THEN
		vTestCases[0].state := utTestCaseStates.ut_PASSED;
		vTestCases[0].msg := 'Parameter act was greater than xp and function returned TRUE -> PASS';
	ELSE
		vTestCases[0].state := utTestCaseStates.ut_FAILED;
		vTestCases[0].msg := 'Parameter act was greater than xp and function returned FALSE -> FAIL';
	END_IF
END_IF
                      
END_ACTION

ACTION TEST_CASE_2_SETUP:
                        IF vTestCases[1].state = utTestCaseStates.ut_SETUP THEN
	(*Setup the test case information*)
	vTestCases[1].id := 2;
    vTestCases[1].desc[0] := 'RETURNS TRUE WHEN PARAMETER ACT EQUAL TO XP';
    vTestCases[1].desc[1] := 'Tests if the function returns True if the parameter act is equal to parameter xp';
	vTestCases[1].desc[2] := 'PASS IF: Return value is TRUE';
	
	(*Setup needed variables*)
	vTestCase2_act := REAL_TO_LREAL(115.4);
	vTestCase2_xp := REAL_TO_LREAL(115.4);
END_IF
                      
END_ACTION

ACTION TEST_CASE_2_EXEC:
                        IF vTestCases[1].state = utTestCaseStates.ut_RUNNING THEN
	(*Run the test case*)
	IF assertGreaterEqual_LREAL(vTestCase2_act, vTestCase2_xp) THEN
		vTestCases[1].state := utTestCaseStates.ut_PASSED;
		vTestCases[1].msg := 'Parameter act was equal to xp and function returned TRUE -> PASS';
	ELSE
		vTestCases[1].state := utTestCaseStates.ut_FAILED;
		vTestCases[1].msg := 'Parameter act was equal to xp and function returned FALSE -> FAIL';
	END_IF
END_IF
                      
END_ACTION

ACTION TEST_CASE_3_SETUP:
                        IF vTestCases[2].state = utTestCaseStates.ut_SETUP THEN
	(*Setup the test case information*)
	vTestCases[2].id := 3;
    vTestCases[2].desc[0] := 'RETURNS FALSE WHEN PARAMETER ACT LESS THAN XP';
    vTestCases[2].desc[1] := 'Tests if the function returns False if the parameter act is less than parameter xp';
	vTestCases[2].desc[2] := 'PASS IF: Return value is FALSE';
	
	(*Setup needed variables*)
	vTestCase3_act := REAL_TO_LREAL(85.4);
	vTestCase3_xp := REAL_TO_LREAL(115.4);
END_IF
                      
END_ACTION

ACTION TEST_CASE_3_EXEC:
                        IF vTestCases[2].state = utTestCaseStates.ut_RUNNING THEN
	(*Run the test case*)
	IF NOT assertGreaterEqual_LREAL(vTestCase3_act, vTestCase3_xp) THEN
		vTestCases[2].state := utTestCaseStates.ut_PASSED;
		vTestCases[2].msg := 'Parameter act was less than xp and function returned FALSE -> PASS';
	ELSE
		vTestCases[2].state := utTestCaseStates.ut_FAILED;
		vTestCases[2].msg := 'Parameter act was less than xp and function returned TRUE -> FAIL';
	END_IF
END_IF
                      
END_ACTION
END_PROGRAM

PROGRAM test_assertGreaterEqual_USINT
  VAR
    vTestCases : ARRAY[0..20] OF utTestCase;  (* Definition of all test cases for this POU *)
    testRunner : utTestSuite;  (* Test Suite fb instance to run the tests *)
    vRunAll : BOOL;  (* Manual command to run all tests for this POU *)
    vResetAll : BOOL;  (* Manual command to reset all tests for this POU *)
    vTestCase1_act : USINT;  (* Test data 1 of test case 1 *)
    vTestCase1_xp : USINT;  (* Test data 2 of test case 1 *)
    vTestCase2_act : USINT;  (* Test data 1 of test case 2 *)
    vTestCase2_xp : USINT;  (* Test data 2 of test case 2 *)
    vTestCase3_act : USINT;  (* Test data 1 of test case 3 *)
    vTestCase3_xp : USINT;  (* Test data 2 of test case 3 *)
  END_VAR

                    (*Run the test cases*)
TEST_CASE_1_SETUP();
TEST_CASE_1_EXEC();

TEST_CASE_2_SETUP();
TEST_CASE_2_EXEC();

TEST_CASE_3_SETUP();
TEST_CASE_3_EXEC();

(*Instantiate the test runner*)
testRunner(
	Id := 77,
	Name := 'assertGreaterEqual_USINT',
    RunTests := GVL.RunAll OR vRunAll,
	ResetTests := GVL.ResetAll OR vResetAll,
	TestCases:=vTestCases);

(*Report the results to the collection global*)
GVL.Results[testRunner.Id] := testRunner.Summary;
                  

ACTION TEST_CASE_1_SETUP:
                        IF vTestCases[0].state = utTestCaseStates.ut_SETUP THEN
	(*Setup the test case information*)
	vTestCases[0].id := 1;
	vTestCases[0].desc[0] := 'RETURNS TRUE WHEN PARAMETER ACT GREATER THAN XP';
    vTestCases[0].desc[1] := 'Tests if the function returns True if the parameter act is greater than parameter xp';
	vTestCases[0].desc[2] := 'PASS IF: Return value is TRUE';
	
	(*Setup needed variables*)
	vTestCase1_act := REAL_TO_USINT(115.4);
	vTestCase1_xp := REAL_TO_USINT(85.4);
END_IF
                      
END_ACTION

ACTION TEST_CASE_1_EXEC:
                        IF vTestCases[0].state = utTestCaseStates.ut_RUNNING THEN
	(*Run the test case*)
	IF assertGreaterEqual_USINT(vTestCase1_act, vTestCase1_xp) THEN
		vTestCases[0].state := utTestCaseStates.ut_PASSED;
		vTestCases[0].msg := 'Parameter act was greater than xp and function returned TRUE -> PASS';
	ELSE
		vTestCases[0].state := utTestCaseStates.ut_FAILED;
		vTestCases[0].msg := 'Parameter act was greater than xp and function returned FALSE -> FAIL';
	END_IF
END_IF
                      
END_ACTION

ACTION TEST_CASE_2_SETUP:
                        IF vTestCases[1].state = utTestCaseStates.ut_SETUP THEN
	(*Setup the test case information*)
	vTestCases[1].id := 2;
    vTestCases[1].desc[0] := 'RETURNS TRUE WHEN PARAMETER ACT EQUAL TO XP';
    vTestCases[1].desc[1] := 'Tests if the function returns True if the parameter act is equal to parameter xp';
	vTestCases[1].desc[2] := 'PASS IF: Return value is TRUE';
	
	(*Setup needed variables*)
	vTestCase2_act := REAL_TO_USINT(115.4);
	vTestCase2_xp := REAL_TO_USINT(115.4);
END_IF
                      
END_ACTION

ACTION TEST_CASE_2_EXEC:
                        IF vTestCases[1].state = utTestCaseStates.ut_RUNNING THEN
	(*Run the test case*)
	IF assertGreaterEqual_USINT(vTestCase2_act, vTestCase2_xp) THEN
		vTestCases[1].state := utTestCaseStates.ut_PASSED;
		vTestCases[1].msg := 'Parameter act was equal to xp and function returned TRUE -> PASS';
	ELSE
		vTestCases[1].state := utTestCaseStates.ut_FAILED;
		vTestCases[1].msg := 'Parameter act was equal to xp and function returned FALSE -> FAIL';
	END_IF
END_IF
                      
END_ACTION

ACTION TEST_CASE_3_SETUP:
                        IF vTestCases[2].state = utTestCaseStates.ut_SETUP THEN
	(*Setup the test case information*)
	vTestCases[2].id := 3;
    vTestCases[2].desc[0] := 'RETURNS FALSE WHEN PARAMETER ACT LESS THAN XP';
    vTestCases[2].desc[1] := 'Tests if the function returns False if the parameter act is less than parameter xp';
	vTestCases[2].desc[2] := 'PASS IF: Return value is FALSE';
	
	(*Setup needed variables*)
	vTestCase3_act := REAL_TO_USINT(85.4);
	vTestCase3_xp := REAL_TO_USINT(115.4);
END_IF
                      
END_ACTION

ACTION TEST_CASE_3_EXEC:
                        IF vTestCases[2].state = utTestCaseStates.ut_RUNNING THEN
	(*Run the test case*)
	IF NOT assertGreaterEqual_USINT(vTestCase3_act, vTestCase3_xp) THEN
		vTestCases[2].state := utTestCaseStates.ut_PASSED;
		vTestCases[2].msg := 'Parameter act was less than xp and function returned FALSE -> PASS';
	ELSE
		vTestCases[2].state := utTestCaseStates.ut_FAILED;
		vTestCases[2].msg := 'Parameter act was less than xp and function returned TRUE -> FAIL';
	END_IF
END_IF
                      
END_ACTION
END_PROGRAM

PROGRAM test_assertGreaterEqual_INT
  VAR
    vTestCases : ARRAY[0..20] OF utTestCase;  (* Definition of all test cases for this POU *)
    testRunner : utTestSuite;  (* Test Suite fb instance to run the tests *)
    vRunAll : BOOL;  (* Manual command to run all tests for this POU *)
    vResetAll : BOOL;  (* Manual command to reset all tests for this POU *)
    vTestCase1_act : INT;  (* Test data 1 of test case 1 *)
    vTestCase1_xp : INT;  (* Test data 2 of test case 1 *)
    vTestCase2_act : INT;  (* Test data 1 of test case 2 *)
    vTestCase2_xp : INT;  (* Test data 2 of test case 2 *)
    vTestCase3_act : INT;  (* Test data 1 of test case 3 *)
    vTestCase3_xp : INT;  (* Test data 2 of test case 3 *)
  END_VAR

                    (*Run the test cases*)
TEST_CASE_1_SETUP();
TEST_CASE_1_EXEC();

TEST_CASE_2_SETUP();
TEST_CASE_2_EXEC();

TEST_CASE_3_SETUP();
TEST_CASE_3_EXEC();

(*Instantiate the test runner*)
testRunner(
	Id := 78,
	Name := 'assertGreaterEqual_INT',
    RunTests := GVL.RunAll OR vRunAll,
	ResetTests := GVL.ResetAll OR vResetAll,
	TestCases:=vTestCases);

(*Report the results to the collection global*)
GVL.Results[testRunner.Id] := testRunner.Summary;
                  

ACTION TEST_CASE_1_SETUP:
                        IF vTestCases[0].state = utTestCaseStates.ut_SETUP THEN
	(*Setup the test case information*)
	vTestCases[0].id := 1;
	vTestCases[0].desc[0] := 'RETURNS TRUE WHEN PARAMETER ACT GREATER THAN XP';
    vTestCases[0].desc[1] := 'Tests if the function returns True if the parameter act is greater than parameter xp';
	vTestCases[0].desc[2] := 'PASS IF: Return value is TRUE';
	
	(*Setup needed variables*)
	vTestCase1_act := REAL_TO_INT(115.4);
	vTestCase1_xp := REAL_TO_INT(85.4);
END_IF
                      
END_ACTION

ACTION TEST_CASE_1_EXEC:
                        IF vTestCases[0].state = utTestCaseStates.ut_RUNNING THEN
	(*Run the test case*)
	IF assertGreaterEqual_INT(vTestCase1_act, vTestCase1_xp) THEN
		vTestCases[0].state := utTestCaseStates.ut_PASSED;
		vTestCases[0].msg := 'Parameter act was greater than xp and function returned TRUE -> PASS';
	ELSE
		vTestCases[0].state := utTestCaseStates.ut_FAILED;
		vTestCases[0].msg := 'Parameter act was greater than xp and function returned FALSE -> FAIL';
	END_IF
END_IF
                      
END_ACTION

ACTION TEST_CASE_2_SETUP:
                        IF vTestCases[1].state = utTestCaseStates.ut_SETUP THEN
	(*Setup the test case information*)
	vTestCases[1].id := 2;
    vTestCases[1].desc[0] := 'RETURNS TRUE WHEN PARAMETER ACT EQUAL TO XP';
    vTestCases[1].desc[1] := 'Tests if the function returns True if the parameter act is equal to parameter xp';
	vTestCases[1].desc[2] := 'PASS IF: Return value is TRUE';
	
	(*Setup needed variables*)
	vTestCase2_act := REAL_TO_INT(115.4);
	vTestCase2_xp := REAL_TO_INT(115.4);
END_IF
                      
END_ACTION

ACTION TEST_CASE_2_EXEC:
                        IF vTestCases[1].state = utTestCaseStates.ut_RUNNING THEN
	(*Run the test case*)
	IF assertGreaterEqual_INT(vTestCase2_act, vTestCase2_xp) THEN
		vTestCases[1].state := utTestCaseStates.ut_PASSED;
		vTestCases[1].msg := 'Parameter act was equal to xp and function returned TRUE -> PASS';
	ELSE
		vTestCases[1].state := utTestCaseStates.ut_FAILED;
		vTestCases[1].msg := 'Parameter act was equal to xp and function returned FALSE -> FAIL';
	END_IF
END_IF
                      
END_ACTION

ACTION TEST_CASE_3_SETUP:
                        IF vTestCases[2].state = utTestCaseStates.ut_SETUP THEN
	(*Setup the test case information*)
	vTestCases[2].id := 3;
    vTestCases[2].desc[0] := 'RETURNS FALSE WHEN PARAMETER ACT LESS THAN XP';
    vTestCases[2].desc[1] := 'Tests if the function returns False if the parameter act is less than parameter xp';
	vTestCases[2].desc[2] := 'PASS IF: Return value is FALSE';
	
	(*Setup needed variables*)
	vTestCase3_act := REAL_TO_INT(85.4);
	vTestCase3_xp := REAL_TO_INT(115.4);
END_IF
                      
END_ACTION

ACTION TEST_CASE_3_EXEC:
                        IF vTestCases[2].state = utTestCaseStates.ut_RUNNING THEN
	(*Run the test case*)
	IF NOT assertGreaterEqual_INT(vTestCase3_act, vTestCase3_xp) THEN
		vTestCases[2].state := utTestCaseStates.ut_PASSED;
		vTestCases[2].msg := 'Parameter act was less than xp and function returned FALSE -> PASS';
	ELSE
		vTestCases[2].state := utTestCaseStates.ut_FAILED;
		vTestCases[2].msg := 'Parameter act was less than xp and function returned TRUE -> FAIL';
	END_IF
END_IF
                      
END_ACTION
END_PROGRAM

PROGRAM test_assertArrayEqual_WSTRING
  VAR
    vTestCases : ARRAY[0..20] OF utTestCase;  (* Definition of all test cases for this POU *)
    testRunner : utTestSuite;  (* Test Suite fb instance to run the tests *)
    vRunAll : BOOL;  (* Manual command to run all tests for this POU *)
    vResetAll : BOOL;  (* Manual command to reset all tests for this POU *)
    vTestCase1_act : ARRAY[0..70] OF WSTRING;  (* Array data 1 of test case 1 *)
    vTestCase1_xp : ARRAY[0..70] OF WSTRING;  (* Array data 2 of test case 1 *)
    vTestCase2_act : ARRAY[0..70] OF WSTRING;  (* Array data 3 of test case 2 *)
    vTestCase2_xp : ARRAY[0..70] OF WSTRING;  (* Array data 4 of test case 2 *)
    i : UINT;  (* Iterator variable i *)
    j : UINT;  (* Iterator variable j *)
  END_VAR

                    (*Run the test cases*)
TEST_CASE_1_SETUP();
TEST_CASE_1_EXEC();

TEST_CASE_2_SETUP();
TEST_CASE_2_EXEC();

(*Instantiate the test runner*)
testRunner(
	Id := 154,
	Name := 'assertArrayEqual_WSTRING',
    RunTests := GVL.RunAll OR vRunAll,
	ResetTests := GVL.ResetAll OR vResetAll,
	TestCases:=vTestCases);

(*Report the results to the collection global*)
GVL.Results[testRunner.Id] := testRunner.Summary;
                  

ACTION TEST_CASE_1_SETUP:
                        IF vTestCases[0].state = utTestCaseStates.ut_SETUP THEN
	(*Setup the test case information*)
	vTestCases[0].id := 1;
	vTestCases[0].desc[0] := 'RETURNS TRUE WHEN ARRAYS EQUAL';
    vTestCases[0].desc[1] := 'Tests if the function returns True if the passed in arrays are identical';
	vTestCases[0].desc[2] := 'PASS IF: Return value is TRUE';
	
	(*Setup needed variables*)
	FOR i:=0 TO 70 DO
		vTestCase1_act[i] := UINT_TO_WSTRING(35 * BOOL_TO_UINT(i MOD 2 = 0));
		vTestCase1_xp[i] := UINT_TO_WSTRING(35 * BOOL_TO_UINT(i MOD 2 = 0));
	END_FOR
END_IF
                      
END_ACTION

ACTION TEST_CASE_1_EXEC:
                        IF vTestCases[0].state = utTestCaseStates.ut_RUNNING THEN
	(*Run the test case*)
	IF assertArrayEqual_WSTRING(ADR(vTestCase1_act), ADR(vTestCase1_xp), SIZEOF(vTestCase1_act)) THEN
		vTestCases[0].state := utTestCaseStates.ut_PASSED;
		vTestCases[0].msg := 'Arrays were equal and function returned TRUE -> PASS';
	ELSE
		vTestCases[0].state := utTestCaseStates.ut_FAILED;
		vTestCases[0].msg := 'Arrays were equal and function returned FALSE -> FAIL';
	END_IF
END_IF
                      
END_ACTION

ACTION TEST_CASE_2_SETUP:
                        IF vTestCases[1].state = utTestCaseStates.ut_SETUP THEN
	(*Setup the test case information*)
	vTestCases[1].id := 2;
	vTestCases[1].desc[0] := 'RETURNS FALSE WHEN ARRAYS NOT EQUAL';
    vTestCases[1].desc[1] := 'Tests if the function returns False if the passed in arrays are not identical';
	vTestCases[1].desc[2] := 'PASS IF: Return value is FALSE';
	
	(*Setup needed variables*)
	FOR j:=0 TO 70 DO
		vTestCase2_act[j] := UINT_TO_WSTRING(35 * BOOL_TO_UINT(j MOD 2 = 0));
		vTestCase2_xp[j] := UINT_TO_WSTRING(35 * BOOL_TO_UINT(j MOD 2 <> 0));
	END_FOR
END_IF
                      
END_ACTION

ACTION TEST_CASE_2_EXEC:
                        IF vTestCases[1].state = utTestCaseStates.ut_RUNNING THEN
	(*Run the test case*)
	IF NOT assertArrayEqual_WSTRING(ADR(vTestCase2_act), ADR(vTestCase2_xp), SIZEOF(vTestCase2_act)) THEN
		vTestCases[1].state := utTestCaseStates.ut_PASSED;
		vTestCases[1].msg := 'Arrays were not equal and function returned FALSE -> PASS';
	ELSE
		vTestCases[1].state := utTestCaseStates.ut_FAILED;
		vTestCases[1].msg := 'Arrays were not equal and function returned TRUE -> FAIL';
	END_IF
END_IF
                      
END_ACTION
END_PROGRAM

PROGRAM test_assertArrayEqual_TIME
  VAR
    vTestCases : ARRAY[0..20] OF utTestCase;  (* Definition of all test cases for this POU *)
    testRunner : utTestSuite;  (* Test Suite fb instance to run the tests *)
    vRunAll : BOOL;  (* Manual command to run all tests for this POU *)
    vResetAll : BOOL;  (* Manual command to reset all tests for this POU *)
    vTestCase1_act : ARRAY[0..70] OF TIME;  (* Array data 1 of test case 1 *)
    vTestCase1_xp : ARRAY[0..70] OF TIME;  (* Array data 2 of test case 1 *)
    vTestCase2_act : ARRAY[0..70] OF TIME;  (* Array data 3 of test case 2 *)
    vTestCase2_xp : ARRAY[0..70] OF TIME;  (* Array data 4 of test case 2 *)
    i : UINT;  (* Iterator variable i *)
    j : UINT;  (* Iterator variable j *)
  END_VAR

                    (*Run the test cases*)
TEST_CASE_1_SETUP();
TEST_CASE_1_EXEC();

TEST_CASE_2_SETUP();
TEST_CASE_2_EXEC();

(*Instantiate the test runner*)
testRunner(
	Id := 155,
	Name := 'assertArrayEqual_TIME',
    RunTests := GVL.RunAll OR vRunAll,
	ResetTests := GVL.ResetAll OR vResetAll,
	TestCases:=vTestCases);

(*Report the results to the collection global*)
GVL.Results[testRunner.Id] := testRunner.Summary;
                  

ACTION TEST_CASE_1_SETUP:
                        IF vTestCases[0].state = utTestCaseStates.ut_SETUP THEN
	(*Setup the test case information*)
	vTestCases[0].id := 1;
	vTestCases[0].desc[0] := 'RETURNS TRUE WHEN ARRAYS EQUAL';
    vTestCases[0].desc[1] := 'Tests if the function returns True if the passed in arrays are identical';
	vTestCases[0].desc[2] := 'PASS IF: Return value is TRUE';
	
	(*Setup needed variables*)
	FOR i:=0 TO 70 DO
		vTestCase1_act[i] := UINT_TO_TIME(35 * BOOL_TO_UINT(i MOD 2 = 0));
		vTestCase1_xp[i] := UINT_TO_TIME(35 * BOOL_TO_UINT(i MOD 2 = 0));
	END_FOR
END_IF
                      
END_ACTION

ACTION TEST_CASE_1_EXEC:
                        IF vTestCases[0].state = utTestCaseStates.ut_RUNNING THEN
	(*Run the test case*)
	IF assertArrayEqual_TIME(ADR(vTestCase1_act), ADR(vTestCase1_xp), SIZEOF(vTestCase1_act)) THEN
		vTestCases[0].state := utTestCaseStates.ut_PASSED;
		vTestCases[0].msg := 'Arrays were equal and function returned TRUE -> PASS';
	ELSE
		vTestCases[0].state := utTestCaseStates.ut_FAILED;
		vTestCases[0].msg := 'Arrays were equal and function returned FALSE -> FAIL';
	END_IF
END_IF
                      
END_ACTION

ACTION TEST_CASE_2_SETUP:
                        IF vTestCases[1].state = utTestCaseStates.ut_SETUP THEN
	(*Setup the test case information*)
	vTestCases[1].id := 2;
	vTestCases[1].desc[0] := 'RETURNS FALSE WHEN ARRAYS NOT EQUAL';
    vTestCases[1].desc[1] := 'Tests if the function returns False if the passed in arrays are not identical';
	vTestCases[1].desc[2] := 'PASS IF: Return value is FALSE';
	
	(*Setup needed variables*)
	FOR j:=0 TO 70 DO
		vTestCase2_act[j] := UINT_TO_TIME(35 * BOOL_TO_UINT(j MOD 2 = 0));
		vTestCase2_xp[j] := UINT_TO_TIME(35 * BOOL_TO_UINT(j MOD 2 <> 0));
	END_FOR
END_IF
                      
END_ACTION

ACTION TEST_CASE_2_EXEC:
                        IF vTestCases[1].state = utTestCaseStates.ut_RUNNING THEN
	(*Run the test case*)
	IF NOT assertArrayEqual_TIME(ADR(vTestCase2_act), ADR(vTestCase2_xp), SIZEOF(vTestCase2_act)) THEN
		vTestCases[1].state := utTestCaseStates.ut_PASSED;
		vTestCases[1].msg := 'Arrays were not equal and function returned FALSE -> PASS';
	ELSE
		vTestCases[1].state := utTestCaseStates.ut_FAILED;
		vTestCases[1].msg := 'Arrays were not equal and function returned TRUE -> FAIL';
	END_IF
END_IF
                      
END_ACTION
END_PROGRAM

PROGRAM test_assertArrayEqual_LDATE_AND_TIME
  VAR
    vTestCases : ARRAY[0..20] OF utTestCase;  (* Definition of all test cases for this POU *)
    testRunner : utTestSuite;  (* Test Suite fb instance to run the tests *)
    vRunAll : BOOL;  (* Manual command to run all tests for this POU *)
    vResetAll : BOOL;  (* Manual command to reset all tests for this POU *)
    vTestCase1_act : ARRAY[0..70] OF LDATE_AND_TIME;  (* Array data 1 of test case 1 *)
    vTestCase1_xp : ARRAY[0..70] OF LDATE_AND_TIME;  (* Array data 2 of test case 1 *)
    vTestCase2_act : ARRAY[0..70] OF LDATE_AND_TIME;  (* Array data 3 of test case 2 *)
    vTestCase2_xp : ARRAY[0..70] OF LDATE_AND_TIME;  (* Array data 4 of test case 2 *)
    i : UINT;  (* Iterator variable i *)
    j : UINT;  (* Iterator variable j *)
  END_VAR

                    (*Run the test cases*)
TEST_CASE_1_SETUP();
TEST_CASE_1_EXEC();

TEST_CASE_2_SETUP();
TEST_CASE_2_EXEC();

(*Instantiate the test runner*)
testRunner(
	Id := 160,
	Name := 'assertArrayEqual_LDATE_AND_TIME',
    RunTests := GVL.RunAll OR vRunAll,
	ResetTests := GVL.ResetAll OR vResetAll,
	TestCases:=vTestCases);

(*Report the results to the collection global*)
GVL.Results[testRunner.Id] := testRunner.Summary;
                  

ACTION TEST_CASE_2_EXEC:
                        IF vTestCases[1].state = utTestCaseStates.ut_RUNNING THEN
	(*Run the test case*)
	IF NOT assertArrayEqual_LDATE_AND_TIME(ADR(vTestCase2_act), ADR(vTestCase2_xp), SIZEOF(vTestCase2_act)) THEN
		vTestCases[1].state := utTestCaseStates.ut_PASSED;
		vTestCases[1].msg := 'Arrays were not equal and function returned FALSE -> PASS';
	ELSE
		vTestCases[1].state := utTestCaseStates.ut_FAILED;
		vTestCases[1].msg := 'Arrays were not equal and function returned TRUE -> FAIL';
	END_IF
END_IF
                      
END_ACTION

ACTION TEST_CASE_1_SETUP:
                        IF vTestCases[0].state = utTestCaseStates.ut_SETUP THEN
	(*Setup the test case information*)
	vTestCases[0].id := 1;
	vTestCases[0].desc[0] := 'RETURNS TRUE WHEN ARRAYS EQUAL';
    vTestCases[0].desc[1] := 'Tests if the function returns True if the passed in arrays are identical';
	vTestCases[0].desc[2] := 'PASS IF: Return value is TRUE';
	
	(*Setup needed variables*)
	FOR i:=0 TO 70 DO
		vTestCase1_act[i] := UINT_TO_LDT(35 * BOOL_TO_UINT(i MOD 2 = 0));
		vTestCase1_xp[i] := UINT_TO_LDT(35 * BOOL_TO_UINT(i MOD 2 = 0));
	END_FOR
END_IF
                      
END_ACTION

ACTION TEST_CASE_1_EXEC:
                        IF vTestCases[0].state = utTestCaseStates.ut_RUNNING THEN
	(*Run the test case*)
	IF assertArrayEqual_LDATE_AND_TIME(ADR(vTestCase1_act), ADR(vTestCase1_xp), SIZEOF(vTestCase1_act)) THEN
		vTestCases[0].state := utTestCaseStates.ut_PASSED;
		vTestCases[0].msg := 'Arrays were equal and function returned TRUE -> PASS';
	ELSE
		vTestCases[0].state := utTestCaseStates.ut_FAILED;
		vTestCases[0].msg := 'Arrays were equal and function returned FALSE -> FAIL';
	END_IF
END_IF
                      
END_ACTION

ACTION TEST_CASE_2_SETUP:
                        IF vTestCases[1].state = utTestCaseStates.ut_SETUP THEN
	(*Setup the test case information*)
	vTestCases[1].id := 2;
	vTestCases[1].desc[0] := 'RETURNS FALSE WHEN ARRAYS NOT EQUAL';
    vTestCases[1].desc[1] := 'Tests if the function returns False if the passed in arrays are not identical';
	vTestCases[1].desc[2] := 'PASS IF: Return value is FALSE';
	
	(*Setup needed variables*)
	FOR j:=0 TO 70 DO
		vTestCase2_act[j] := UINT_TO_LDT(35 * BOOL_TO_UINT(j MOD 2 = 0));
		vTestCase2_xp[j] := UINT_TO_LDT(35 * BOOL_TO_UINT(j MOD 2 <> 0));
	END_FOR
END_IF
                      
END_ACTION
END_PROGRAM

PROGRAM test_assertArrayEqual_TIME_OF_DAY
  VAR
    vTestCases : ARRAY[0..20] OF utTestCase;  (* Definition of all test cases for this POU *)
    testRunner : utTestSuite;  (* Test Suite fb instance to run the tests *)
    vRunAll : BOOL;  (* Manual command to run all tests for this POU *)
    vResetAll : BOOL;  (* Manual command to reset all tests for this POU *)
    vTestCase1_act : ARRAY[0..70] OF TOD;  (* Array data 1 of test case 1 *)
    vTestCase1_xp : ARRAY[0..70] OF TOD;  (* Array data 2 of test case 1 *)
    vTestCase2_act : ARRAY[0..70] OF TOD;  (* Array data 3 of test case 2 *)
    vTestCase2_xp : ARRAY[0..70] OF TOD;  (* Array data 4 of test case 2 *)
    i : UINT;  (* Iterator variable i *)
    j : UINT;  (* Iterator variable j *)
  END_VAR

                    (*Run the test cases*)
TEST_CASE_1_SETUP();
TEST_CASE_1_EXEC();

TEST_CASE_2_SETUP();
TEST_CASE_2_EXEC();

(*Instantiate the test runner*)
testRunner(
	Id := 161,
	Name := 'assertArrayEqual_TIME_OF_DAY',
    RunTests := GVL.RunAll OR vRunAll,
	ResetTests := GVL.ResetAll OR vResetAll,
	TestCases:=vTestCases);

(*Report the results to the collection global*)
GVL.Results[testRunner.Id] := testRunner.Summary;
                  

ACTION TEST_CASE_1_SETUP:
                        IF vTestCases[0].state = utTestCaseStates.ut_SETUP THEN
	(*Setup the test case information*)
	vTestCases[0].id := 1;
	vTestCases[0].desc[0] := 'RETURNS TRUE WHEN ARRAYS EQUAL';
    vTestCases[0].desc[1] := 'Tests if the function returns True if the passed in arrays are identical';
	vTestCases[0].desc[2] := 'PASS IF: Return value is TRUE';
	
	(*Setup needed variables*)
	FOR i:=0 TO 70 DO
		vTestCase1_act[i] := UINT_TO_TOD(35 * BOOL_TO_UINT(i MOD 2 = 0));
		vTestCase1_xp[i] := UINT_TO_TOD(35 * BOOL_TO_UINT(i MOD 2 = 0));
	END_FOR
END_IF
                      
END_ACTION

ACTION TEST_CASE_1_EXEC:
                        IF vTestCases[0].state = utTestCaseStates.ut_RUNNING THEN
	(*Run the test case*)
	IF assertArrayEqual_TIME_OF_DAY(ADR(vTestCase1_act), ADR(vTestCase1_xp), SIZEOF(vTestCase1_act)) THEN
		vTestCases[0].state := utTestCaseStates.ut_PASSED;
		vTestCases[0].msg := 'Arrays were equal and function returned TRUE -> PASS';
	ELSE
		vTestCases[0].state := utTestCaseStates.ut_FAILED;
		vTestCases[0].msg := 'Arrays were equal and function returned FALSE -> FAIL';
	END_IF
END_IF
                      
END_ACTION

ACTION TEST_CASE_2_SETUP:
                        IF vTestCases[1].state = utTestCaseStates.ut_SETUP THEN
	(*Setup the test case information*)
	vTestCases[1].id := 2;
	vTestCases[1].desc[0] := 'RETURNS FALSE WHEN ARRAYS NOT EQUAL';
    vTestCases[1].desc[1] := 'Tests if the function returns False if the passed in arrays are not identical';
	vTestCases[1].desc[2] := 'PASS IF: Return value is FALSE';
	
	(*Setup needed variables*)
	FOR j:=0 TO 70 DO
		vTestCase2_act[j] := UINT_TO_TOD(35 * BOOL_TO_UINT(j MOD 2 = 0));
		vTestCase2_xp[j] := UINT_TO_TOD(35 * BOOL_TO_UINT(j MOD 2 <> 0));
	END_FOR
END_IF
                      
END_ACTION

ACTION TEST_CASE_2_EXEC:
                        IF vTestCases[1].state = utTestCaseStates.ut_RUNNING THEN
	(*Run the test case*)
	IF NOT assertArrayEqual_TIME_OF_DAY(ADR(vTestCase2_act), ADR(vTestCase2_xp), SIZEOF(vTestCase2_act)) THEN
		vTestCases[1].state := utTestCaseStates.ut_PASSED;
		vTestCases[1].msg := 'Arrays were not equal and function returned FALSE -> PASS';
	ELSE
		vTestCases[1].state := utTestCaseStates.ut_FAILED;
		vTestCases[1].msg := 'Arrays were not equal and function returned TRUE -> FAIL';
	END_IF
END_IF
                      
END_ACTION
END_PROGRAM

PROGRAM test_assertArrayEqual_LTIME_OF_DAY
  VAR
    vTestCases : ARRAY[0..20] OF utTestCase;  (* Definition of all test cases for this POU *)
    testRunner : utTestSuite;  (* Test Suite fb instance to run the tests *)
    vRunAll : BOOL;  (* Manual command to run all tests for this POU *)
    vResetAll : BOOL;  (* Manual command to reset all tests for this POU *)
    vTestCase1_act : ARRAY[0..70] OF LTIME_OF_DAY;  (* Array data 1 of test case 1 *)
    vTestCase1_xp : ARRAY[0..70] OF LTIME_OF_DAY;  (* Array data 2 of test case 1 *)
    vTestCase2_act : ARRAY[0..70] OF LTIME_OF_DAY;  (* Array data 3 of test case 2 *)
    vTestCase2_xp : ARRAY[0..70] OF LTIME_OF_DAY;  (* Array data 4 of test case 2 *)
    i : UINT;  (* Iterator variable i *)
    j : UINT;  (* Iterator variable j *)
  END_VAR

                    (*Run the test cases*)
TEST_CASE_1_SETUP();
TEST_CASE_1_EXEC();

TEST_CASE_2_SETUP();
TEST_CASE_2_EXEC();

(*Instantiate the test runner*)
testRunner(
	Id := 162,
	Name := 'assertArrayEqual_LTIME_OF_DAY',
    RunTests := GVL.RunAll OR vRunAll,
	ResetTests := GVL.ResetAll OR vResetAll,
	TestCases:=vTestCases);

(*Report the results to the collection global*)
GVL.Results[testRunner.Id] := testRunner.Summary;
                  

ACTION TEST_CASE_1_SETUP:
                        IF vTestCases[0].state = utTestCaseStates.ut_SETUP THEN
	(*Setup the test case information*)
	vTestCases[0].id := 1;
	vTestCases[0].desc[0] := 'RETURNS TRUE WHEN ARRAYS EQUAL';
    vTestCases[0].desc[1] := 'Tests if the function returns True if the passed in arrays are identical';
	vTestCases[0].desc[2] := 'PASS IF: Return value is TRUE';
	
	(*Setup needed variables*)
	FOR i:=0 TO 70 DO
		vTestCase1_act[i] := UINT_TO_LTOD(35 * BOOL_TO_UINT(i MOD 2 = 0));
		vTestCase1_xp[i] := UINT_TO_LTOD(35 * BOOL_TO_UINT(i MOD 2 = 0));
	END_FOR
END_IF
                      
END_ACTION

ACTION TEST_CASE_1_EXEC:
                        IF vTestCases[0].state = utTestCaseStates.ut_RUNNING THEN
	(*Run the test case*)
	IF assertArrayEqual_LTIME_OF_DAY(ADR(vTestCase1_act), ADR(vTestCase1_xp), SIZEOF(vTestCase1_act)) THEN
		vTestCases[0].state := utTestCaseStates.ut_PASSED;
		vTestCases[0].msg := 'Arrays were equal and function returned TRUE -> PASS';
	ELSE
		vTestCases[0].state := utTestCaseStates.ut_FAILED;
		vTestCases[0].msg := 'Arrays were equal and function returned FALSE -> FAIL';
	END_IF
END_IF
                      
END_ACTION

ACTION TEST_CASE_2_SETUP:
                        IF vTestCases[1].state = utTestCaseStates.ut_SETUP THEN
	(*Setup the test case information*)
	vTestCases[1].id := 2;
	vTestCases[1].desc[0] := 'RETURNS FALSE WHEN ARRAYS NOT EQUAL';
    vTestCases[1].desc[1] := 'Tests if the function returns False if the passed in arrays are not identical';
	vTestCases[1].desc[2] := 'PASS IF: Return value is FALSE';
	
	(*Setup needed variables*)
	FOR j:=0 TO 70 DO
		vTestCase2_act[j] := UINT_TO_LTOD(35 * BOOL_TO_UINT(j MOD 2 = 0));
		vTestCase2_xp[j] := UINT_TO_LTOD(35 * BOOL_TO_UINT(j MOD 2 <> 0));
	END_FOR
END_IF
                      
END_ACTION

ACTION TEST_CASE_2_EXEC:
                        IF vTestCases[1].state = utTestCaseStates.ut_RUNNING THEN
	(*Run the test case*)
	IF NOT assertArrayEqual_LTIME_OF_DAY(ADR(vTestCase2_act), ADR(vTestCase2_xp), SIZEOF(vTestCase2_act)) THEN
		vTestCases[1].state := utTestCaseStates.ut_PASSED;
		vTestCases[1].msg := 'Arrays were not equal and function returned FALSE -> PASS';
	ELSE
		vTestCases[1].state := utTestCaseStates.ut_FAILED;
		vTestCases[1].msg := 'Arrays were not equal and function returned TRUE -> FAIL';
	END_IF
END_IF
                      
END_ACTION
END_PROGRAM

PROGRAM test_assertArrayEqual_DATE_AND_TIME
  VAR
    vTestCases : ARRAY[0..20] OF utTestCase;  (* Definition of all test cases for this POU *)
    testRunner : utTestSuite;  (* Test Suite fb instance to run the tests *)
    vRunAll : BOOL;  (* Manual command to run all tests for this POU *)
    vResetAll : BOOL;  (* Manual command to reset all tests for this POU *)
    vTestCase1_act : ARRAY[0..70] OF DT;  (* Array data 1 of test case 1 *)
    vTestCase1_xp : ARRAY[0..70] OF DT;  (* Array data 2 of test case 1 *)
    vTestCase2_act : ARRAY[0..70] OF DT;  (* Array data 3 of test case 2 *)
    vTestCase2_xp : ARRAY[0..70] OF DT;  (* Array data 4 of test case 2 *)
    i : UINT;  (* Iterator variable i *)
    j : UINT;  (* Iterator variable j *)
  END_VAR

                    (*Run the test cases*)
TEST_CASE_1_SETUP();
TEST_CASE_1_EXEC();

TEST_CASE_2_SETUP();
TEST_CASE_2_EXEC();

(*Instantiate the test runner*)
testRunner(
	Id := 159,
	Name := 'assertArrayEqual_DATE_AND_TIME',
    RunTests := GVL.RunAll OR vRunAll,
	ResetTests := GVL.ResetAll OR vResetAll,
	TestCases:=vTestCases);

(*Report the results to the collection global*)
GVL.Results[testRunner.Id] := testRunner.Summary;
                  

ACTION TEST_CASE_1_EXEC:
                        IF vTestCases[0].state = utTestCaseStates.ut_RUNNING THEN
	(*Run the test case*)
	IF assertArrayEqual_DATE_AND_TIME(ADR(vTestCase1_act), ADR(vTestCase1_xp), SIZEOF(vTestCase1_act)) THEN
		vTestCases[0].state := utTestCaseStates.ut_PASSED;
		vTestCases[0].msg := 'Arrays were equal and function returned TRUE -> PASS';
	ELSE
		vTestCases[0].state := utTestCaseStates.ut_FAILED;
		vTestCases[0].msg := 'Arrays were equal and function returned FALSE -> FAIL';
	END_IF
END_IF
                      
END_ACTION

ACTION TEST_CASE_2_SETUP:
                        IF vTestCases[1].state = utTestCaseStates.ut_SETUP THEN
	(*Setup the test case information*)
	vTestCases[1].id := 2;
	vTestCases[1].desc[0] := 'RETURNS FALSE WHEN ARRAYS NOT EQUAL';
    vTestCases[1].desc[1] := 'Tests if the function returns False if the passed in arrays are not identical';
	vTestCases[1].desc[2] := 'PASS IF: Return value is FALSE';
	
	(*Setup needed variables*)
	FOR j:=0 TO 70 DO
		vTestCase2_act[j] := UINT_TO_DT(35 * BOOL_TO_UINT(j MOD 2 = 0));
		vTestCase2_xp[j] := UINT_TO_DT(35 * BOOL_TO_UINT(j MOD 2 <> 0));
	END_FOR
END_IF
                      
END_ACTION

ACTION TEST_CASE_2_EXEC:
                        IF vTestCases[1].state = utTestCaseStates.ut_RUNNING THEN
	(*Run the test case*)
	IF NOT assertArrayEqual_DATE_AND_TIME(ADR(vTestCase2_act), ADR(vTestCase2_xp), SIZEOF(vTestCase2_act)) THEN
		vTestCases[1].state := utTestCaseStates.ut_PASSED;
		vTestCases[1].msg := 'Arrays were not equal and function returned FALSE -> PASS';
	ELSE
		vTestCases[1].state := utTestCaseStates.ut_FAILED;
		vTestCases[1].msg := 'Arrays were not equal and function returned TRUE -> FAIL';
	END_IF
END_IF
                      
END_ACTION

ACTION TEST_CASE_1_SETUP:
                        IF vTestCases[0].state = utTestCaseStates.ut_SETUP THEN
	(*Setup the test case information*)
	vTestCases[0].id := 1;
	vTestCases[0].desc[0] := 'RETURNS TRUE WHEN ARRAYS EQUAL';
    vTestCases[0].desc[1] := 'Tests if the function returns True if the passed in arrays are identical';
	vTestCases[0].desc[2] := 'PASS IF: Return value is TRUE';
	
	(*Setup needed variables*)
	FOR i:=0 TO 70 DO
		vTestCase1_act[i] := UINT_TO_DT(35 * BOOL_TO_UINT(i MOD 2 = 0));
		vTestCase1_xp[i] := UINT_TO_DT(35 * BOOL_TO_UINT(i MOD 2 = 0));
	END_FOR
END_IF
                      
END_ACTION
END_PROGRAM

PROGRAM test_assertArrayEqual_LTIME
  VAR
    vTestCases : ARRAY[0..20] OF utTestCase;  (* Definition of all test cases for this POU *)
    testRunner : utTestSuite;  (* Test Suite fb instance to run the tests *)
    vRunAll : BOOL;  (* Manual command to run all tests for this POU *)
    vResetAll : BOOL;  (* Manual command to reset all tests for this POU *)
    vTestCase1_act : ARRAY[0..70] OF LTIME;  (* Array data 1 of test case 1 *)
    vTestCase1_xp : ARRAY[0..70] OF LTIME;  (* Array data 2 of test case 1 *)
    vTestCase2_act : ARRAY[0..70] OF LTIME;  (* Array data 3 of test case 2 *)
    vTestCase2_xp : ARRAY[0..70] OF LTIME;  (* Array data 4 of test case 2 *)
    i : UINT;  (* Iterator variable i *)
    j : UINT;  (* Iterator variable j *)
  END_VAR

                    (*Run the test cases*)
TEST_CASE_1_SETUP();
TEST_CASE_1_EXEC();

TEST_CASE_2_SETUP();
TEST_CASE_2_EXEC();

(*Instantiate the test runner*)
testRunner(
	Id := 156,
	Name := 'assertArrayEqual_LTIME',
    RunTests := GVL.RunAll OR vRunAll,
	ResetTests := GVL.ResetAll OR vResetAll,
	TestCases:=vTestCases);

(*Report the results to the collection global*)
GVL.Results[testRunner.Id] := testRunner.Summary;
                  

ACTION TEST_CASE_2_SETUP:
                        IF vTestCases[1].state = utTestCaseStates.ut_SETUP THEN
	(*Setup the test case information*)
	vTestCases[1].id := 2;
	vTestCases[1].desc[0] := 'RETURNS FALSE WHEN ARRAYS NOT EQUAL';
    vTestCases[1].desc[1] := 'Tests if the function returns False if the passed in arrays are not identical';
	vTestCases[1].desc[2] := 'PASS IF: Return value is FALSE';
	
	(*Setup needed variables*)
	FOR j:=0 TO 70 DO
		vTestCase2_act[j] := UINT_TO_LTIME(35 * BOOL_TO_UINT(j MOD 2 = 0));
		vTestCase2_xp[j] := UINT_TO_LTIME(35 * BOOL_TO_UINT(j MOD 2 <> 0));
	END_FOR
END_IF
                      
END_ACTION

ACTION TEST_CASE_1_SETUP:
                        IF vTestCases[0].state = utTestCaseStates.ut_SETUP THEN
	(*Setup the test case information*)
	vTestCases[0].id := 1;
	vTestCases[0].desc[0] := 'RETURNS TRUE WHEN ARRAYS EQUAL';
    vTestCases[0].desc[1] := 'Tests if the function returns True if the passed in arrays are identical';
	vTestCases[0].desc[2] := 'PASS IF: Return value is TRUE';
	
	(*Setup needed variables*)
	FOR i:=0 TO 70 DO
		vTestCase1_act[i] := UINT_TO_LTIME(35 * BOOL_TO_UINT(i MOD 2 = 0));
		vTestCase1_xp[i] := UINT_TO_LTIME(35 * BOOL_TO_UINT(i MOD 2 = 0));
	END_FOR
END_IF
                      
END_ACTION

ACTION TEST_CASE_1_EXEC:
                        IF vTestCases[0].state = utTestCaseStates.ut_RUNNING THEN
	(*Run the test case*)
	IF assertArrayEqual_LTIME(ADR(vTestCase1_act), ADR(vTestCase1_xp), SIZEOF(vTestCase1_act)) THEN
		vTestCases[0].state := utTestCaseStates.ut_PASSED;
		vTestCases[0].msg := 'Arrays were equal and function returned TRUE -> PASS';
	ELSE
		vTestCases[0].state := utTestCaseStates.ut_FAILED;
		vTestCases[0].msg := 'Arrays were equal and function returned FALSE -> FAIL';
	END_IF
END_IF
                      
END_ACTION

ACTION TEST_CASE_2_EXEC:
                        IF vTestCases[1].state = utTestCaseStates.ut_RUNNING THEN
	(*Run the test case*)
	IF NOT assertArrayEqual_LTIME(ADR(vTestCase2_act), ADR(vTestCase2_xp), SIZEOF(vTestCase2_act)) THEN
		vTestCases[1].state := utTestCaseStates.ut_PASSED;
		vTestCases[1].msg := 'Arrays were not equal and function returned FALSE -> PASS';
	ELSE
		vTestCases[1].state := utTestCaseStates.ut_FAILED;
		vTestCases[1].msg := 'Arrays were not equal and function returned TRUE -> FAIL';
	END_IF
END_IF
                      
END_ACTION
END_PROGRAM

PROGRAM test_assertTrue
  VAR
    vTestCases : ARRAY[0..20] OF utTestCase;  (* Definition of all test cases for this POU *)
    testRunner : utTestSuite;  (* Test Suite fb instance to run the tests *)
    vRunAll : BOOL;  (* Manual command to run all tests for this POU *)
    vResetAll : BOOL;  (* Manual command to reset all tests for this POU *)
    vTestCase1_act : BOOL;  (* Test data 1 of test case 1 *)
    vTestCase2_act : BOOL;  (* Test data 1 of test case 2 *)
  END_VAR

                    (*Run the test cases*)
TEST_CASE_1_SETUP();
TEST_CASE_1_EXEC();

TEST_CASE_2_SETUP();
TEST_CASE_2_EXEC();

(*Instantiate the test runner*)
testRunner(
	Id := 163,
	Name := 'assertTrue',
    RunTests := GVL.RunAll OR vRunAll,
	ResetTests := GVL.ResetAll OR vResetAll,
	TestCases:=vTestCases);

(*Report the results to the collection global*)
GVL.Results[testRunner.Id] := testRunner.Summary;
                  

ACTION TEST_CASE_2_SETUP:
                        IF vTestCases[1].state = utTestCaseStates.ut_SETUP THEN
	(*Setup the test case information*)
	vTestCases[1].id := 2;
    vTestCases[1].desc[0] := 'RETURNS FALSE WHEN CONDITION IS FALSE';
    vTestCases[1].desc[1] := 'Tests if the function returns False if the condition is FALSE';
	vTestCases[1].desc[2] := 'PASS IF: Return value is FALSE';
	
	(*Setup needed variables*)
	vTestCase2_act := FALSE;
END_IF
                      
END_ACTION

ACTION TEST_CASE_1_SETUP:
                        IF vTestCases[0].state = utTestCaseStates.ut_SETUP THEN
	(*Setup the test case information*)
	vTestCases[0].id := 1;
	vTestCases[0].desc[0] := 'RETURNS TRUE WHEN CONDITION TRUE';
    vTestCases[0].desc[1] := 'Tests if the function returns True if the condition is TRUE';
	vTestCases[0].desc[2] := 'PASS IF: Return value is TRUE';
	
	(*Setup needed variables*)
	vTestCase1_act := TRUE;
END_IF
                      
END_ACTION

ACTION TEST_CASE_1_EXEC:
                        IF vTestCases[0].state = utTestCaseStates.ut_RUNNING THEN
	(*Run the test case*)
	IF assertTrue(vTestCase1_act) THEN
		vTestCases[0].state := utTestCaseStates.ut_PASSED;
		vTestCases[0].msg := 'Condition was True and function returned TRUE -> PASS';
	ELSE
		vTestCases[0].state := utTestCaseStates.ut_FAILED;
		vTestCases[0].msg := 'Condition was True and function returned FALSE -> FAIL';
	END_IF
END_IF
                      
END_ACTION

ACTION TEST_CASE_2_EXEC:
                        IF vTestCases[1].state = utTestCaseStates.ut_RUNNING THEN
	(*Run the test case*)
	IF NOT assertTrue(vTestCase2_act) THEN
		vTestCases[1].state := utTestCaseStates.ut_PASSED;
		vTestCases[1].msg := 'Condition was False and function returned FALSE -> PASS';
	ELSE
		vTestCases[1].state := utTestCaseStates.ut_FAILED;
		vTestCases[1].msg := 'Condition was False and function returned TRUE -> FAIL';
	END_IF
END_IF
                      
END_ACTION
END_PROGRAM

PROGRAM test_assertArrayEqual_DATE
  VAR
    vTestCases : ARRAY[0..20] OF utTestCase;  (* Definition of all test cases for this POU *)
    testRunner : utTestSuite;  (* Test Suite fb instance to run the tests *)
    vRunAll : BOOL;  (* Manual command to run all tests for this POU *)
    vResetAll : BOOL;  (* Manual command to reset all tests for this POU *)
    vTestCase1_act : ARRAY[0..70] OF DATE;  (* Array data 1 of test case 1 *)
    vTestCase1_xp : ARRAY[0..70] OF DATE;  (* Array data 2 of test case 1 *)
    vTestCase2_act : ARRAY[0..70] OF DATE;  (* Array data 3 of test case 2 *)
    vTestCase2_xp : ARRAY[0..70] OF DATE;  (* Array data 4 of test case 2 *)
    i : UINT;  (* Iterator variable i *)
    j : UINT;  (* Iterator variable j *)
  END_VAR

                    (*Run the test cases*)
TEST_CASE_1_SETUP();
TEST_CASE_1_EXEC();

TEST_CASE_2_SETUP();
TEST_CASE_2_EXEC();

(*Instantiate the test runner*)
testRunner(
	Id := 157,
	Name := 'assertArrayEqual_DATE',
    RunTests := GVL.RunAll OR vRunAll,
	ResetTests := GVL.ResetAll OR vResetAll,
	TestCases:=vTestCases);

(*Report the results to the collection global*)
GVL.Results[testRunner.Id] := testRunner.Summary;
                  

ACTION TEST_CASE_1_SETUP:
                        IF vTestCases[0].state = utTestCaseStates.ut_SETUP THEN
	(*Setup the test case information*)
	vTestCases[0].id := 1;
	vTestCases[0].desc[0] := 'RETURNS TRUE WHEN ARRAYS EQUAL';
    vTestCases[0].desc[1] := 'Tests if the function returns True if the passed in arrays are identical';
	vTestCases[0].desc[2] := 'PASS IF: Return value is TRUE';
	
	(*Setup needed variables*)
	FOR i:=0 TO 70 DO
		vTestCase1_act[i] := UINT_TO_DATE(35 * BOOL_TO_UINT(i MOD 2 = 0));
		vTestCase1_xp[i] := UINT_TO_DATE(35 * BOOL_TO_UINT(i MOD 2 = 0));
	END_FOR
END_IF
                      
END_ACTION

ACTION TEST_CASE_1_EXEC:
                        IF vTestCases[0].state = utTestCaseStates.ut_RUNNING THEN
	(*Run the test case*)
	IF assertArrayEqual_DATE(ADR(vTestCase1_act), ADR(vTestCase1_xp), SIZEOF(vTestCase1_act)) THEN
		vTestCases[0].state := utTestCaseStates.ut_PASSED;
		vTestCases[0].msg := 'Arrays were equal and function returned TRUE -> PASS';
	ELSE
		vTestCases[0].state := utTestCaseStates.ut_FAILED;
		vTestCases[0].msg := 'Arrays were equal and function returned FALSE -> FAIL';
	END_IF
END_IF
                      
END_ACTION

ACTION TEST_CASE_2_SETUP:
                        IF vTestCases[1].state = utTestCaseStates.ut_SETUP THEN
	(*Setup the test case information*)
	vTestCases[1].id := 2;
	vTestCases[1].desc[0] := 'RETURNS FALSE WHEN ARRAYS NOT EQUAL';
    vTestCases[1].desc[1] := 'Tests if the function returns False if the passed in arrays are not identical';
	vTestCases[1].desc[2] := 'PASS IF: Return value is FALSE';
	
	(*Setup needed variables*)
	FOR j:=0 TO 70 DO
		vTestCase2_act[j] := UINT_TO_DATE(35 * BOOL_TO_UINT(j MOD 2 = 0));
		vTestCase2_xp[j] := UINT_TO_DATE(35 * BOOL_TO_UINT(j MOD 2 <> 0));
	END_FOR
END_IF
                      
END_ACTION

ACTION TEST_CASE_2_EXEC:
                        IF vTestCases[1].state = utTestCaseStates.ut_RUNNING THEN
	(*Run the test case*)
	IF NOT assertArrayEqual_DATE(ADR(vTestCase2_act), ADR(vTestCase2_xp), SIZEOF(vTestCase2_act)) THEN
		vTestCases[1].state := utTestCaseStates.ut_PASSED;
		vTestCases[1].msg := 'Arrays were not equal and function returned FALSE -> PASS';
	ELSE
		vTestCases[1].state := utTestCaseStates.ut_FAILED;
		vTestCases[1].msg := 'Arrays were not equal and function returned TRUE -> FAIL';
	END_IF
END_IF
                      
END_ACTION
END_PROGRAM

PROGRAM test_assertFalse
  VAR
    vTestCases : ARRAY[0..20] OF utTestCase;  (* Definition of all test cases for this POU *)
    testRunner : utTestSuite;  (* Test Suite fb instance to run the tests *)
    vRunAll : BOOL;  (* Manual command to run all tests for this POU *)
    vResetAll : BOOL;  (* Manual command to reset all tests for this POU *)
    vTestCase1_act : BOOL;  (* Test data 1 of test case 1 *)
    vTestCase2_act : BOOL;  (* Test data 1 of test case 2 *)
  END_VAR

                    (*Run the test cases*)
TEST_CASE_1_SETUP();
TEST_CASE_1_EXEC();

TEST_CASE_2_SETUP();
TEST_CASE_2_EXEC();

(*Instantiate the test runner*)
testRunner(
	Id := 164,
	Name := 'assertFalse',
    RunTests := GVL.RunAll OR vRunAll,
	ResetTests := GVL.ResetAll OR vResetAll,
	TestCases:=vTestCases);

(*Report the results to the collection global*)
GVL.Results[testRunner.Id] := testRunner.Summary;
                  

ACTION TEST_CASE_1_SETUP:
                        IF vTestCases[0].state = utTestCaseStates.ut_SETUP THEN
	(*Setup the test case information*)
	vTestCases[0].id := 1;
	vTestCases[0].desc[0] := 'RETURNS TRUE WHEN CONDITION FALSE';
    vTestCases[0].desc[1] := 'Tests if the function returns True if the condition is FALSE';
	vTestCases[0].desc[2] := 'PASS IF: Return value is TRUE';
	
	(*Setup needed variables*)
	vTestCase1_act := FALSE;
END_IF
                      
END_ACTION

ACTION TEST_CASE_1_EXEC:
                        IF vTestCases[0].state = utTestCaseStates.ut_RUNNING THEN
	(*Run the test case*)
	IF assertFalse(vTestCase1_act) THEN
		vTestCases[0].state := utTestCaseStates.ut_PASSED;
		vTestCases[0].msg := 'Condition was False and function returned TRUE -> PASS';
	ELSE
		vTestCases[0].state := utTestCaseStates.ut_FAILED;
		vTestCases[0].msg := 'Condition was False and function returned FALSE -> FAIL';
	END_IF
END_IF
                      
END_ACTION

ACTION TEST_CASE_2_SETUP:
                        IF vTestCases[1].state = utTestCaseStates.ut_SETUP THEN
	(*Setup the test case information*)
	vTestCases[1].id := 2;
    vTestCases[1].desc[0] := 'RETURNS FALSE WHEN CONDITION IS TRUE';
    vTestCases[1].desc[1] := 'Tests if the function returns False if the condition is TRUE';
	vTestCases[1].desc[2] := 'PASS IF: Return value is FALSE';
	
	(*Setup needed variables*)
	vTestCase2_act := TRUE;
END_IF
                      
END_ACTION

ACTION TEST_CASE_2_EXEC:
                        IF vTestCases[1].state = utTestCaseStates.ut_RUNNING THEN
	(*Run the test case*)
	IF NOT assertFalse(vTestCase2_act) THEN
		vTestCases[1].state := utTestCaseStates.ut_PASSED;
		vTestCases[1].msg := 'Condition was True and function returned FALSE -> PASS';
	ELSE
		vTestCases[1].state := utTestCaseStates.ut_FAILED;
		vTestCases[1].msg := 'Condition was True and function returned TRUE -> FAIL';
	END_IF
END_IF
                      
END_ACTION
END_PROGRAM

PROGRAM test_assertLessEqual_DINT
  VAR
    vTestCases : ARRAY[0..20] OF utTestCase;  (* Definition of all test cases for this POU *)
    testRunner : utTestSuite;  (* Test Suite fb instance to run the tests *)
    vRunAll : BOOL;  (* Manual command to run all tests for this POU *)
    vResetAll : BOOL;  (* Manual command to reset all tests for this POU *)
    vTestCase1_act : DINT;  (* Test data 1 of test case 1 *)
    vTestCase1_xp : DINT;  (* Test data 2 of test case 1 *)
    vTestCase2_act : DINT;  (* Test data 1 of test case 2 *)
    vTestCase2_xp : DINT;  (* Test data 2 of test case 2 *)
    vTestCase3_act : DINT;  (* Test data 1 of test case 3 *)
    vTestCase3_xp : DINT;  (* Test data 2 of test case 3 *)
  END_VAR

                    (*Run the test cases*)
TEST_CASE_1_SETUP();
TEST_CASE_1_EXEC();

TEST_CASE_2_SETUP();
TEST_CASE_2_EXEC();

TEST_CASE_3_SETUP();
TEST_CASE_3_EXEC();

(*Instantiate the test runner*)
testRunner(
	Id := 124,
	Name := 'assertLessEqual_DINT',
    RunTests := GVL.RunAll OR vRunAll,
	ResetTests := GVL.ResetAll OR vResetAll,
	TestCases:=vTestCases);

(*Report the results to the collection global*)
GVL.Results[testRunner.Id] := testRunner.Summary;
                  

ACTION TEST_CASE_1_EXEC:
                        IF vTestCases[0].state = utTestCaseStates.ut_RUNNING THEN
	(*Run the test case*)
	IF assertLessEqual_DINT(vTestCase1_act, vTestCase1_xp) THEN
		vTestCases[0].state := utTestCaseStates.ut_PASSED;
		vTestCases[0].msg := 'Parameter act was less than xp and function returned TRUE -> PASS';
	ELSE
		vTestCases[0].state := utTestCaseStates.ut_FAILED;
		vTestCases[0].msg := 'Parameter act was less than xp and function returned FALSE -> FAIL';
	END_IF
END_IF
                      
END_ACTION

ACTION TEST_CASE_3_SETUP:
                        IF vTestCases[2].state = utTestCaseStates.ut_SETUP THEN
	(*Setup the test case information*)
	vTestCases[2].id := 3;
    vTestCases[2].desc[0] := 'RETURNS FALSE WHEN PARAMETER ACT GREATER THAN XP';
    vTestCases[2].desc[1] := 'Tests if the function returns False if the parameter act is greater than parameter xp';
	vTestCases[2].desc[2] := 'PASS IF: Return value is FALSE';
	
	(*Setup needed variables*)
	vTestCase3_act := REAL_TO_DINT(115.4);
	vTestCase3_xp := REAL_TO_DINT(85.4);
END_IF
                      
END_ACTION

ACTION TEST_CASE_3_EXEC:
                        IF vTestCases[2].state = utTestCaseStates.ut_RUNNING THEN
	(*Run the test case*)
	IF NOT assertLessEqual_DINT(vTestCase3_act, vTestCase3_xp) THEN
		vTestCases[2].state := utTestCaseStates.ut_PASSED;
		vTestCases[2].msg := 'Parameter act was greater than xp and function returned FALSE -> PASS';
	ELSE
		vTestCases[2].state := utTestCaseStates.ut_FAILED;
		vTestCases[2].msg := 'Parameter act was greater than xp and function returned TRUE -> FAIL';
	END_IF
END_IF
                      
END_ACTION

ACTION TEST_CASE_1_SETUP:
                        IF vTestCases[0].state = utTestCaseStates.ut_SETUP THEN
	(*Setup the test case information*)
	vTestCases[0].id := 1;
	vTestCases[0].desc[0] := 'RETURNS TRUE WHEN PARAMETER ACT LESS THAN XP';
    vTestCases[0].desc[1] := 'Tests if the function returns True if the parameter act is less than parameter xp';
	vTestCases[0].desc[2] := 'PASS IF: Return value is TRUE';
	
	(*Setup needed variables*)
	vTestCase1_act := REAL_TO_DINT(85.4);
	vTestCase1_xp := REAL_TO_DINT(115.4);
END_IF
                      
END_ACTION

ACTION TEST_CASE_2_SETUP:
                        IF vTestCases[1].state = utTestCaseStates.ut_SETUP THEN
	(*Setup the test case information*)
	vTestCases[1].id := 2;
    vTestCases[1].desc[0] := 'RETURNS TRUE WHEN PARAMETER ACT EQUAL TO XP';
    vTestCases[1].desc[1] := 'Tests if the function returns True if the parameter act is equal to parameter xp';
	vTestCases[1].desc[2] := 'PASS IF: Return value is TRUE';
	
	(*Setup needed variables*)
	vTestCase2_act := REAL_TO_DINT(115.4);
	vTestCase2_xp := REAL_TO_DINT(115.4);
END_IF
                      
END_ACTION

ACTION TEST_CASE_2_EXEC:
                        IF vTestCases[1].state = utTestCaseStates.ut_RUNNING THEN
	(*Run the test case*)
	IF assertLessEqual_DINT(vTestCase2_act, vTestCase2_xp) THEN
		vTestCases[1].state := utTestCaseStates.ut_PASSED;
		vTestCases[1].msg := 'Parameter act was equal to xp and function returned TRUE -> PASS';
	ELSE
		vTestCases[1].state := utTestCaseStates.ut_FAILED;
		vTestCases[1].msg := 'Parameter act was equal to xp and function returned FALSE -> FAIL';
	END_IF
END_IF
                      
END_ACTION
END_PROGRAM

PROGRAM test_assertArrayEqual_STRING
  VAR
    vTestCases : ARRAY[0..20] OF utTestCase;  (* Definition of all test cases for this POU *)
    testRunner : utTestSuite;  (* Test Suite fb instance to run the tests *)
    vRunAll : BOOL;  (* Manual command to run all tests for this POU *)
    vResetAll : BOOL;  (* Manual command to reset all tests for this POU *)
    vTestCase1_act : ARRAY[0..70] OF STRING;  (* Array data 1 of test case 1 *)
    vTestCase1_xp : ARRAY[0..70] OF STRING;  (* Array data 2 of test case 1 *)
    vTestCase2_act : ARRAY[0..70] OF STRING;  (* Array data 3 of test case 2 *)
    vTestCase2_xp : ARRAY[0..70] OF STRING;  (* Array data 4 of test case 2 *)
    i : UINT;  (* Iterator variable i *)
    j : UINT;  (* Iterator variable j *)
  END_VAR

                    (*Run the test cases*)
TEST_CASE_1_SETUP();
TEST_CASE_1_EXEC();

TEST_CASE_2_SETUP();
TEST_CASE_2_EXEC();

(*Instantiate the test runner*)
testRunner(
	Id := 153,
	Name := 'assertArrayEqual_STRING',
    RunTests := GVL.RunAll OR vRunAll,
	ResetTests := GVL.ResetAll OR vResetAll,
	TestCases:=vTestCases);

(*Report the results to the collection global*)
GVL.Results[testRunner.Id] := testRunner.Summary;
                  

ACTION TEST_CASE_2_EXEC:
                        IF vTestCases[1].state = utTestCaseStates.ut_RUNNING THEN
	(*Run the test case*)
	IF NOT assertArrayEqual_STRING(ADR(vTestCase2_act), ADR(vTestCase2_xp), SIZEOF(vTestCase2_act)) THEN
		vTestCases[1].state := utTestCaseStates.ut_PASSED;
		vTestCases[1].msg := 'Arrays were not equal and function returned FALSE -> PASS';
	ELSE
		vTestCases[1].state := utTestCaseStates.ut_FAILED;
		vTestCases[1].msg := 'Arrays were not equal and function returned TRUE -> FAIL';
	END_IF
END_IF
                      
END_ACTION

ACTION TEST_CASE_1_SETUP:
                        IF vTestCases[0].state = utTestCaseStates.ut_SETUP THEN
	(*Setup the test case information*)
	vTestCases[0].id := 1;
	vTestCases[0].desc[0] := 'RETURNS TRUE WHEN ARRAYS EQUAL';
    vTestCases[0].desc[1] := 'Tests if the function returns True if the passed in arrays are identical';
	vTestCases[0].desc[2] := 'PASS IF: Return value is TRUE';
	
	(*Setup needed variables*)
	FOR i:=0 TO 70 DO
		vTestCase1_act[i] := UINT_TO_STRING(35 * BOOL_TO_UINT(i MOD 2 = 0));
		vTestCase1_xp[i] := UINT_TO_STRING(35 * BOOL_TO_UINT(i MOD 2 = 0));
	END_FOR
END_IF
                      
END_ACTION

ACTION TEST_CASE_1_EXEC:
                        IF vTestCases[0].state = utTestCaseStates.ut_RUNNING THEN
	(*Run the test case*)
	IF assertArrayEqual_STRING(ADR(vTestCase1_act), ADR(vTestCase1_xp), SIZEOF(vTestCase1_act)) THEN
		vTestCases[0].state := utTestCaseStates.ut_PASSED;
		vTestCases[0].msg := 'Arrays were equal and function returned TRUE -> PASS';
	ELSE
		vTestCases[0].state := utTestCaseStates.ut_FAILED;
		vTestCases[0].msg := 'Arrays were equal and function returned FALSE -> FAIL';
	END_IF
END_IF
                      
END_ACTION

ACTION TEST_CASE_2_SETUP:
                        IF vTestCases[1].state = utTestCaseStates.ut_SETUP THEN
	(*Setup the test case information*)
	vTestCases[1].id := 2;
	vTestCases[1].desc[0] := 'RETURNS FALSE WHEN ARRAYS NOT EQUAL';
    vTestCases[1].desc[1] := 'Tests if the function returns False if the passed in arrays are not identical';
	vTestCases[1].desc[2] := 'PASS IF: Return value is FALSE';
	
	(*Setup needed variables*)
	FOR j:=0 TO 70 DO
		vTestCase2_act[j] := UINT_TO_STRING(35 * BOOL_TO_UINT(j MOD 2 = 0));
		vTestCase2_xp[j] := UINT_TO_STRING(35 * BOOL_TO_UINT(j MOD 2 <> 0));
	END_FOR
END_IF
                      
END_ACTION
END_PROGRAM

PROGRAM test_assertLessEqual_LREAL
  VAR
    vTestCases : ARRAY[0..20] OF utTestCase;  (* Definition of all test cases for this POU *)
    testRunner : utTestSuite;  (* Test Suite fb instance to run the tests *)
    vRunAll : BOOL;  (* Manual command to run all tests for this POU *)
    vResetAll : BOOL;  (* Manual command to reset all tests for this POU *)
    vTestCase1_act : LREAL;  (* Test data 1 of test case 1 *)
    vTestCase1_xp : LREAL;  (* Test data 2 of test case 1 *)
    vTestCase2_act : LREAL;  (* Test data 1 of test case 2 *)
    vTestCase2_xp : LREAL;  (* Test data 2 of test case 2 *)
    vTestCase3_act : LREAL;  (* Test data 1 of test case 3 *)
    vTestCase3_xp : LREAL;  (* Test data 2 of test case 3 *)
  END_VAR

                    (*Run the test cases*)
TEST_CASE_1_SETUP();
TEST_CASE_1_EXEC();

TEST_CASE_2_SETUP();
TEST_CASE_2_EXEC();

TEST_CASE_3_SETUP();
TEST_CASE_3_EXEC();

(*Instantiate the test runner*)
testRunner(
	Id := 129,
	Name := 'assertLessEqual_LREAL',
    RunTests := GVL.RunAll OR vRunAll,
	ResetTests := GVL.ResetAll OR vResetAll,
	TestCases:=vTestCases);

(*Report the results to the collection global*)
GVL.Results[testRunner.Id] := testRunner.Summary;
                  

ACTION TEST_CASE_3_SETUP:
                        IF vTestCases[2].state = utTestCaseStates.ut_SETUP THEN
	(*Setup the test case information*)
	vTestCases[2].id := 3;
    vTestCases[2].desc[0] := 'RETURNS FALSE WHEN PARAMETER ACT GREATER THAN XP';
    vTestCases[2].desc[1] := 'Tests if the function returns False if the parameter act is greater than parameter xp';
	vTestCases[2].desc[2] := 'PASS IF: Return value is FALSE';
	
	(*Setup needed variables*)
	vTestCase3_act := REAL_TO_LREAL(115.4);
	vTestCase3_xp := REAL_TO_LREAL(85.4);
END_IF
                      
END_ACTION

ACTION TEST_CASE_3_EXEC:
                        IF vTestCases[2].state = utTestCaseStates.ut_RUNNING THEN
	(*Run the test case*)
	IF NOT assertLessEqual_LREAL(vTestCase3_act, vTestCase3_xp) THEN
		vTestCases[2].state := utTestCaseStates.ut_PASSED;
		vTestCases[2].msg := 'Parameter act was greater than xp and function returned FALSE -> PASS';
	ELSE
		vTestCases[2].state := utTestCaseStates.ut_FAILED;
		vTestCases[2].msg := 'Parameter act was greater than xp and function returned TRUE -> FAIL';
	END_IF
END_IF
                      
END_ACTION

ACTION TEST_CASE_1_SETUP:
                        IF vTestCases[0].state = utTestCaseStates.ut_SETUP THEN
	(*Setup the test case information*)
	vTestCases[0].id := 1;
	vTestCases[0].desc[0] := 'RETURNS TRUE WHEN PARAMETER ACT LESS THAN XP';
    vTestCases[0].desc[1] := 'Tests if the function returns True if the parameter act is less than parameter xp';
	vTestCases[0].desc[2] := 'PASS IF: Return value is TRUE';
	
	(*Setup needed variables*)
	vTestCase1_act := REAL_TO_LREAL(85.4);
	vTestCase1_xp := REAL_TO_LREAL(115.4);
END_IF
                      
END_ACTION

ACTION TEST_CASE_1_EXEC:
                        IF vTestCases[0].state = utTestCaseStates.ut_RUNNING THEN
	(*Run the test case*)
	IF assertLessEqual_LREAL(vTestCase1_act, vTestCase1_xp) THEN
		vTestCases[0].state := utTestCaseStates.ut_PASSED;
		vTestCases[0].msg := 'Parameter act was less than xp and function returned TRUE -> PASS';
	ELSE
		vTestCases[0].state := utTestCaseStates.ut_FAILED;
		vTestCases[0].msg := 'Parameter act was less than xp and function returned FALSE -> FAIL';
	END_IF
END_IF
                      
END_ACTION

